// SIMATIC STEP 7 (V5.x) project 0715-19068
// CPU: CPU 315-2 DP
// CPU: CPU 313C
// station: Hardware
// station: Rigid stranding 61/630
// station: P_ADR_BUS
// station: P_ADR_BUS
// station: Hardware
// station: Loader_Cage6_12_18_24
// program: S7 Program
// program: Programma S7
// program: MASTERDRIVES VC(CUVC)
// program: MASTERDRIVES VC(CUVC)
// program: MASTERDRIVES VC(CUVC)
// program: MASTERDRIVES VC(CUVC)
// program: MASTERDRIVES VC(CUVC)
// program: MASTERDRIVES VC(CUVC)
// program: MASTERDRIVES VC(CUVC)
// program: MASTERDRIVES VC(CUVC)
// program: MASTERDRIVES VC(CUVC)
// program: MASTERDRIVES VC(CUVC)

SYMBOL_TABLE
"Drives --> Plc"	DB 1	DB 1	// Drive --> Plc Data Block
"Plc --> Drives"	DB 2	DB 2	// Plc --> Drive Data Block
"Profibus SFC Alarm"	DB 3	DB 3	// Profibus SFC Alarm Data Block
"Take-up traverse"	DB 5	DB 5	// Take-up traverse Data Block
"Take-up"	DB 7	DB 7	// Take-up data block
"Capstan"	DB 9	DB 9	// Capstan data block
"Cage 24"	DB 15	DB 15	// Cage 24 data block
"Cage 24 preforming"	DB 18	DB 18	// Cage 24 preforming data block
"Cage 18"	DB 20	DB 20	// Cage 18 data block
"Cage 18 preforming"	DB 23	DB 23	// Cage 18 preforming data block
"Cage 12"	DB 25	DB 25	// Cage 12 data block
"Cage 12 preforming"	DB 28	DB 28	// Cage 12 preforming data block
"Cage 6"	DB 30	DB 30	// Cage 6 data block
"Pay-off 630"	DB 35	DB 35	// Pay-off 630 data block
"Metercounter"	DB 41	DB 41	// Metercounter data block
"Line"	DB 55	DB 55	// Line data block
"HMI animation"	DB 60	DB 60	// HMI animation data block
"MAP_DI"	DB 91	DB 91	// DIGITAL INPUT MAP
"MAP_DO"	DB 93	DB 93	// DIGITAL OUTPUT MAP
"Db Plc <=> HMI"	DB 100	DB 100	// Db Plc <=> HMI data block
"Count setting"	DB 101	DB 101	// Count setting data block
"FB125"	DB 125	FB 125	// FB125 data block
"DETAIL_DP_DIAG"	FB 125	FB 125
"Alarms Reset"	FC 1	FC 1	// Alarms reset function
"Profibus alarms"	FC 2	FC 2	// Profibus alarms function
"Profibus unit"	FC 3	FC 3	// Profibus unit function
"Take-up traverse alarms"	FC 4	FC 4	// Take-up traverse alarms function
"Take-up traverse unit"	FC 5	FC 5	// Take-up traverse unit function
"Take-up alarms"	FC 6	FC 6	// Take-up alarms function
"Take-up unit"	FC 7	FC 7	// Take-up unit function
"Capstan alarms"	FC 8	FC 8	// Capstan alarms function
"Capstan unit"	FC 9	FC 9	// Capstan unit function
"Door Cage Lock"	FC 10	FC 10	// Door Cage Lock
"Cage common function"	FC 13	FC 13	// Cage common function
"Cage 24 alarms"	FC 14	FC 14	// Cage 24 alarms function
"Cage 24 unit"	FC 15	FC 15	// Cage 24 unit function
"Cage 24 loading fase"	FC 16	FC 16	// Cage 24 loading fase function
"Cage 24 preforming alarm"	FC 17	FC 17	// Cage 24 preforming alarms function
"Cage 24 preforming unit"	FC 18	FC 18	// Cage 24 preforming unit function
"Cage 18 alarms"	FC 19	FC 19	// Cage 18 alarms function
"Cage 18 unit"	FC 20	FC 20	// Cage 18 unit function
"Cage 18 loading fase"	FC 21	FC 21	// Cage 18 loading fase function
"Cage 18 preforming alarm"	FC 22	FC 22	// Cage 18 preforming alarms function
"Cage 18 preforming unit"	FC 23	FC 23	// Cage 18 preforming unit function
"Cage 12 alarms"	FC 24	FC 24	// Cage 12 alarms function
"Cage 12 unit"	FC 25	FC 25	// Cage 12 unit function
"Cage 12 loading fase"	FC 26	FC 26	// Cage 12 loading fase function
"Cage 12 preforming alarm"	FC 27	FC 27	// Cage 12 preforming alarms function
"Cage 12 preforming unit"	FC 28	FC 28	// Cage 12 preforming unit function
"Cage 6 alarms"	FC 29	FC 29	// Cage 6 alarms function
"Cage 6 unit"	FC 30	FC 30	// Cage 6 unit function
"Cage 6 loading fase"	FC 31	FC 31	// Cage 6 loading fase function
"Cage 6 preforming alarms"	FC 32	FC 32	// Cage 6 preforming alarms function
"Cage 6 preforming unit"	FC 33	FC 33	// Cage 6 preforming unit function
"Pay-off 630 alarms"	FC 34	FC 34	// Pay-off 630 alarms function
"Pay-off 630 unit"	FC 35	FC 35	// Pay-off 630 unit function
"Metercounter alarms"	FC 40	FC 40	// Metercounter alarms function
"Metercounter unit"	FC 41	FC 41	// Metercounter unit function
"Common function"	FC 50	FC 50	// Common function
"Hour counter"	FC 51	FC 51	// Hour counter function
"Line alarms"	FC 52	FC 52	// Line alarms function
"Line unit"	FC 53	FC 53	// Line unit function
"Run consent"	FC 54	FC 54	// Run consents function
"Line jog - line run"	FC 55	FC 55	// Line jog - line run function
"Line reference"	FC 56	FC 56	// Line reference function
"Linear speed"	FC 57	FC 57	// Linear speed function
"Missing power supply"	FC 59	FC 59	// Missing power supply function
"HMI animation unit"	FC 60	FC 60	// HMI animation function
"Take-up traverse impulse"	FC 61	FC 61	// Take-up traverse impulses function
"Cage 24 wires insertion"	FC 70	FC 70	// Cage 24 wires insertion function
"Cage 18 wires insertion"	FC 71	FC 71	// Cage 18 wires insertion function
"Cage 12 wires insertion"	FC 72	FC 72	// Cage 12 wires insertion function
"Cage 6 wires insertion"	FC 73	FC 73	// Cage 6 wires insertion function
"Wires break time"	FC 74	FC 74	// Wires break time function
"Bobbins diameter"	FC 79	FC 79	// Bobbins diameter
"Bobbins brake"	FC 80	FC 80	// Bobbins brake
"Rpm increase"	FC 81	FC 81	// Rpm increase
"Map Input Function"	FC 91	FC 91	// Map Input Function
"Map Output Function"	FC 93	FC 93	// Map Output Function
"Increase-decrease"	FC 100	FC 100	// Increase-decrease function
"Flip-Flop"	FC 101	FC 101	// Flip-flop function
"Ramp"	FC 102	FC 102	// Ramp function
"16 Bit Filter"	FC 103	FC 103	// 16 Bit filter function
"Diameter calculation"	FC 105	FC 105	// Diameter calculation function
"Increase-decrease head"	FC 106	FC 106	// Increase-decrease head function
"32 Bit filter"	FC 108	FC 108	// 32 Bit filter function
"Capstan linear speed"	FC 112	FC 112	// Capstan linear speed function
"Bobbins wire management"	FC 113	FC 113	// Bobbins wire management function
"Bobbin diameter calculat"	FC 114	FC 114	// Bobbin diameter calculaton function
"Motor status HMI"	FC 115	FC 115	// Motor status checking for HMI animation function
"Rotation control"	FC 200	FC 200	// Rotation control function
"-126K1:Auxiliary"	I 0.0	BOOL	// Auxiliary on
"-126K4"	I 0.1	BOOL	// Emergency push-buttons
"-175S3"	I 0.2	BOOL	// Cabinet thermo-switch
"-112Q3"	I 0.3	BOOL	// Auxiliary 220v transformer overload
"-108G1:Alarm"	I 0.4	BOOL	// 24DC UPS module battery alarm
"-108G1:Bat ok"	I 0.5	BOOL	// 24DC UPS module battery packs ok
"-116Q1"	I 0.6	BOOL	// Cabinet air fans overload
"E000.7"	I 0.7	BOOL	// Spare
"-119Q1"	I 1.0	BOOL	// Dryer supply overload
"-141R1:T2"	I 1.1	BOOL	// Ac motor drives feeder braking resistor alarm
"-140G1:X104:20"	I 1.2	BOOL	// Ac motor drives feeder dc bus alarm
"-922S3"	I 1.3	BOOL	// Take-up traverse quick left push-buttons main panel
"-922S4"	I 1.4	BOOL	// Take-up traverse quick right push-buttons main panel
"-112Q8"	I 1.5	BOOL	// Take-up 220vac power supply overload
"-109Q7"	I 1.6	BOOL	// Take-up 24vdc power supply overload
"-922S5"	I 1.7	BOOL	// Take-up bobbin increase pull push-button
"-922S6"	I 2.0	BOOL	// Take-up bobbin decrease pull push-button
"-922S7"	I 2.1	BOOL	// Take-up bobbin stop push-buttons
"-922S8"	I 2.2	BOOL	// Take-up bobbin run push-buttons
"-705Q1"	I 2.3	BOOL	// Capstan motor blower overload
"-718S4"	I 2.4	BOOL	// Capstan minimum air pressure pressure-switch
"-718S5"	I 2.5	BOOL	// Capstan motor brake control pressure-switch
"-718B6"	I 2.6	BOOL	// Capstan cable clock open sensor
"-177S6"	I 2.7	BOOL	// Cable block opening selector-switch
"-177S7:Forward"	I 3.0	BOOL	// Capstan forward jog selector-switch
"-177S7:Backward"	I 3.1	BOOL	// Capstan backward jog selector-switch
"-540Q1"	I 3.2	BOOL	// Cage 18 230vac power supply overload
"-109Q11"	I 3.3	BOOL	// Cage 18 24vdc power supply overload
"-505Q2"	I 3.4	BOOL	// Cage 18 loading motor overload
"-505Q1"	I 3.5	BOOL	// Cage 18 motor blower overload
"-507Q2"	I 3.6	BOOL	// Cage 18 preforming motor electric brake overload
"-507Q1"	I 3.7	BOOL	// Cage 18 preforming motor blower overload
"E004.0"	I 4.0	BOOL	// Spare
"-506Q1"	I 4.1	BOOL	// Cage 18 guard blower motor overload
"-440Q1"	I 4.2	BOOL	// Cage 12 230vac power supply overload
"-109Q10"	I 4.3	BOOL	// Cage 12 24vdc power supply overload
"-405Q2"	I 4.4	BOOL	// Cage 12 loading motor overload
"-405Q1"	I 4.5	BOOL	// Cage 12 motor blower overload
"-407Q2"	I 4.6	BOOL	// Cage 12 preforming motor electric brake overload
"-407Q1"	I 4.7	BOOL	// Cage 12 preforming motor blower overload
"E005.0"	I 5.0	BOOL	// Spare
"-406Q1"	I 5.1	BOOL	// Cage 12 guard blower motor overload
"-340Q1"	I 5.2	BOOL	// Cage 6 230vac power supply overload
"-109Q9"	I 5.3	BOOL	// Cage 6 24vdc power supply overload
"-305Q2"	I 5.4	BOOL	// Cage 6 loading motor overload
"-305Q1"	I 5.5	BOOL	// Cage 6 motor blower overload
"E005.6"	I 5.6	BOOL	// Spare
"-306Q1"	I 5.7	BOOL	// Cage 6 guard blower motor overload
"E006.0"	I 6.0	BOOL	// Spare
"E006.1"	I 6.1	BOOL	// Spare
"E006.2"	I 6.2	BOOL	// Spare
"-177S1"	I 6.3	BOOL	// Line stop push-buttons
"-177S2"	I 6.4	BOOL	// Line run push-buttons
"-177S3"	I 6.5	BOOL	// Line jog push-buttons
"-177S4"	I 6.6	BOOL	// Line alarms reset push-buttons
"-177S5"	I 6.7	BOOL	// Hold line speed push-button
"-640Q1"	I 7.0	BOOL	// Cage 24 230VAC supply overload
"-109Q12"	I 7.1	BOOL	// Cage 24 24VDC supply overload
"-605Q2"	I 7.2	BOOL	// Cage 24 loading motor overload
"-605Q1"	I 7.3	BOOL	// Cage 24 motor blower overload
"-607Q2"	I 7.4	BOOL	// Cage 24 preforming motor electric brake overload
"-607Q1"	I 7.5	BOOL	// Cage 24 preforming motor blower overload
"E007.6"	I 7.6	BOOL	// Spare
"-606Q1"	I 7.7	BOOL	// Cage 24 guard  blower motor overload
"-112K1"	I 8.0	BOOL	// Power supply on
"-112K1:66"	I 8.1	BOOL	// Power supply on end of time
"-113G1:4"	I 8.2	BOOL	// 230VAC UPS main failure
"-113G1:3"	I 8.3	BOOL	// 230VAC UPS battery nearly low
"-109Q6"	I 8.4	BOOL	// 24DC aux. feeding overload
"-115Q1"	I 8.5	BOOL	// preforming motor blower and inverter fan supply overload
"-140Q1"	I 8.6	BOOL	// AC motor drive feeder fan overload
"-109Q2"	I 8.7	BOOL	// 24VDC PLC input supply overload
"+MCB06:7"	I 9.0	BOOL	// Cage 6 Loader in stand by zone
"+MCB06:8"	I 9.1	BOOL	// Cage 6 Loader inside cage
"+MCB06:9"	I 9.2	BOOL	// Cage 6 Loader open clamp
"+MCB06:10"	I 9.3	BOOL	// Cage 6 Loader to parcking zone
"+MCB12:7"	I 9.4	BOOL	// Cage 12 Loader in stand by zone
"+MCB12:8"	I 9.5	BOOL	// Cage 12 Loader inside cage
"+MCB12:9"	I 9.6	BOOL	// Cage 12 Loader open clamp
"+MCB12:10"	I 9.7	BOOL	// Cage 12 Loader to parcking zone
"+MCB18:7"	I 10.0	BOOL	// Cage 18 Loader in stand by zone
"+MCB18:8"	I 10.1	BOOL	// Cage 18 Loader inside cage
"+MCB18:9"	I 10.2	BOOL	// Cage 18 Loader open clamp
"+MCB18:10"	I 10.3	BOOL	// Cage 18 Loader to parcking zone
"+MCB24:7"	I 10.4	BOOL	// Cage 24 Loader in stand by zone
"+MCB24:8"	I 10.5	BOOL	// Cage 24 Loader inside cage
"+MCB24:9"	I 10.6	BOOL	// Cage 24 Loader open clamp
"+MCB24:10"	I 10.7	BOOL	// Cage 24 Loader to parcking zone
"E011.0"	I 11.0	BOOL	// Spare
"E011.1"	I 11.1	BOOL	// Spare
"E011.2"	I 11.2	BOOL	// Spare
"E011.3"	I 11.3	BOOL	// Spare
"E011.4"	I 11.4	BOOL	// Spare
"E011.5"	I 11.5	BOOL	// Spare
"E011.6"	I 11.6	BOOL	// Spare
"E011.7"	I 11.7	BOOL	// Spare
"-961S1"	I 32.0	BOOL	// Take-up idle pintle up limit-switch
"-961S2"	I 32.1	BOOL	// Take-up idle pintle down limit-switch
"-961S3"	I 32.2	BOOL	// Take-up driven pintle up limit-switch
"-961S4"	I 32.3	BOOL	// Take-up driven pintle down limit-switch
"-961S5:UP"	I 33.0	BOOL	// Take-up driven pintle up selector-switch
"-961S5:DOWN"	I 33.1	BOOL	// Take-up driven pintle down selector-switch
"-961S7:UP"	I 33.2	BOOL	// Take-up idle pintle up selector-switch
"-961S7:DOWN"	I 33.3	BOOL	// Take-up idle pintle down selector-switch
"-962S1:UP"	I 34.0	BOOL	// Take-up pintles up selector-switches
"-962S1:DOWN"	I 34.1	BOOL	// Take-up pintles down selector-switches
"-962S3:OPEN"	I 34.2	BOOL	// Take-up idle pintle opening selector-switches
"-962S3:CLOSE"	I 34.3	BOOL	// Take-up idle pintle closing selector-switches
"-962S5"	I 35.0	BOOL	// Take-up idle pintle emergency limit-switch
"-962S6"	I 35.1	BOOL	// Take-up driven pintle emergency limit-switch
"-962S7"	I 35.2	BOOL	// Take-up traverse quick left push-buttons local panel
"-962S8"	I 35.3	BOOL	// Take-up traverse quick right push-buttons local panel
"-964S1:Forward"	I 36.0	BOOL	// Take-up bobbin forward jog selector-switch
"-964S1:Backward"	I 36.1	BOOL	// Take-up bobbin backward jog selector-switch
"-964B3"	I 36.2	BOOL	// Take-up traverse translation zero point sensor
"-964B4"	I 36.3	BOOL	// Take-up traverse inversion delay sensor
"-941Q2"	I 37.0	BOOL	// Take-up bobbin motor electric brake overload
"-945Q2"	I 37.1	BOOL	// Take-up traverse motor blower overload
"-944Q1"	I 37.2	BOOL	// Take-up ac motors overload
"-945Q1"	I 37.3	BOOL	// Take-up bobbin motor blower overload
"-661S1"	I 42.0	BOOL	// Cage 24 loading line presence of air pressure-switch
"-661S2"	I 42.1	BOOL	// Cage 24 brake control pressure-switch
"-661S3"	I 42.2	BOOL	// Cage 24 minimum air pressure pressure-switch
"-661S4"	I 42.3	BOOL	// Cage 24 piston engaged into cage limit-switch
"-661S5"	I 42.4	BOOL	// Cage 24 piston disingaged out of cage limit-switch
"-661S6"	I 42.5	BOOL	// Cage 24 loading motor engaged sensor
"-661S7"	I 42.6	BOOL	// Cage 24 loading motor disengaged sensor
"-661S8"	I 42.7	BOOL	// Cage 24 air pipe  limit-switch
"-662B1"	I 43.0	BOOL	// Cage 24 presence of bobbin photocell -loading-
"-662B2"	I 43.1	BOOL	// Cage 24 loading stop photocell
"-662S3"	I 43.2	BOOL	// Cage 24 break of wire from ring
"-686Y1"	I 43.3	BOOL	// Cage 24 front door limit-switch
"-662S5"	I 43.4	BOOL	// Cage 24 rear door limit-switches
"-662S6"	I 43.5	BOOL	// Cage 24 front guard open limit-switch
"-662B7"	I 43.6	BOOL	// Cage 24 front guard closed sensor
"-662B8"	I 43.7	BOOL	// Cage 24 guard presence of man photocell
"-663S1"	I 44.0	BOOL	// Cage 24 line stop push-button
"-663S2"	I 44.1	BOOL	// Cage 24 line jog push-button
"-663S3"	I 44.2	BOOL	// Cage 24 loading run push-button
"-663S4"	I 44.3	BOOL	// Cage 24 alarms reset push-button
"-663S5:CLOSING"	I 44.4	BOOL	// Cage 24 guard closing selector-switch
"-663S5:OPENING"	I 44.5	BOOL	// Cage 24 guard opening selector-switch
"-663S7:CLOSING"	I 44.6	BOOL	// Cage 24 pintles closing selector-switch
"-663S7:OPENING"	I 44.7	BOOL	// Cage 24 pintles opening selector-switch
"-664S1:CLOSING"	I 45.0	BOOL	// Cage 24 pintles locking system closing selector-switch
"-664S1:OPENING"	I 45.1	BOOL	// Cage 24 pintles locking system opening selector-switch
"E045.2"	I 45.2	BOOL	// Spare
"E045.3"	I 45.3	BOOL	// Spare
"E045.4"	I 45.4	BOOL	// Spare
"E045.5"	I 45.5	BOOL	// Spare
"-664S7"	I 45.6	BOOL	// Cage 24 loading insertion push-button
"E045.7"	I 45.7	BOOL	// Spare
"E046.0"	I 46.0	BOOL	// Spare
"E046.1"	I 46.1	BOOL	// Spare
"E046.2"	I 46.2	BOOL	// Spare
"E046.3"	I 46.3	BOOL	// Spare
"E046.4"	I 46.4	BOOL	// Spare
"E046.5"	I 46.5	BOOL	// Spare
"-688Y8"	I 46.6	BOOL	// Cage 24 preforming guard limit-switch
"-665S8"	I 46.7	BOOL	// Cage 24 preforming brake release push-button
"-666S1"	I 47.0	BOOL	// Cage 24 preforming line stop push-button
"-666S2"	I 47.1	BOOL	// Cage 24 preforming line jog push-button
"-667B1"	I 47.2	BOOL	// Cage 24 bobbin 1 break of wire and diameter calculation
"-667B2"	I 47.3	BOOL	// Cage 24 bobbin 2 break of wire
"-667B3"	I 47.4	BOOL	// Cage 24 bobbin 3 break of wire
"-667B4"	I 47.5	BOOL	// Cage 24 bobbin 4 break of wire
"-667B5"	I 47.6	BOOL	// Cage 24 bobbin 5 break of wire
"-667B6"	I 47.7	BOOL	// Cage 24 bobbin 6 break of wire
"-667B7"	I 48.0	BOOL	// Cage 24 bobbin 7 break of wire
"-667B8"	I 48.1	BOOL	// Cage 24 bobbin 8 break of wire
"-668B1"	I 48.2	BOOL	// Cage 24 bobbin 9 break of wire
"-668B2"	I 48.3	BOOL	// Cage 24 bobbin 10 break of wire
"-668B3"	I 48.4	BOOL	// Cage 24 bobbin 11 break of wire
"-668B4"	I 48.5	BOOL	// Cage 24 bobbin 12 break of wire
"-668B5"	I 48.6	BOOL	// Cage 24 bobbin 13 break of wire
"-668B6"	I 48.7	BOOL	// Cage 24 bobbin 14 break of wire
"-668B7"	I 49.0	BOOL	// Cage 24 bobbin 15 break of wire
"-668B8"	I 49.1	BOOL	// Cage 24 bobbin 16 break of wire
"-669B1"	I 49.2	BOOL	// Cage 24 bobbin 17 break of wire
"-669B2"	I 49.3	BOOL	// Cage 24 bobbin 18 break of wire
"-669B3"	I 49.4	BOOL	// Cage 24 bobbin 19 break of wire
"-669B4"	I 49.5	BOOL	// Cage 24 bobbin 20 break of wire
"-669B5"	I 49.6	BOOL	// Cage 24 bobbin 21 break of wire
"-669B6"	I 49.7	BOOL	// Cage 24 bobbin 22 break of wire
"-669B7"	I 50.0	BOOL	// Cage 24 bobbin 23 break of wire
"-669B8"	I 50.1	BOOL	// Cage 24 bobbin 24 break of wire
"-670S1"	I 50.2	BOOL	// Cage 24 bobbin brakes air tank pressure switch
"-670S2"	I 50.3	BOOL	// Cage 24 line 1 pintles open
"-670S3"	I 50.4	BOOL	// Cage 24 line 2 pintles open
"-670S4"	I 50.5	BOOL	// Cage 24 line 3 pintles open
"E050.6"	I 50.6	BOOL	// Spare
"E050.7"	I 50.7	BOOL	// Spare
"E051.0"	I 51.0	BOOL	// Spare
"E051.1"	I 51.1	BOOL	// Spare
"E051.2"	I 51.2	BOOL	// Spare
"E051.3"	I 51.3	BOOL	// Spare
"E051.4"	I 51.4	BOOL	// Spare
"E051.5"	I 51.5	BOOL	// Spare
"E051.6"	I 51.6	BOOL	// Spare
"E051.7"	I 51.7	BOOL	// Spare
"-561S1"	I 52.0	BOOL	// Cage 18 loading line presence of air pressure-switch
"-561S2"	I 52.1	BOOL	// Cage 18 brake control pressure-switch
"-561S3"	I 52.2	BOOL	// Cage 18 minimum air pressure pressure-switch
"-561S4"	I 52.3	BOOL	// Cage 18 piston engaged in cage limit-switch
"-561S5"	I 52.4	BOOL	// Cage 18 piston disengaged from cage limit-switch
"-561B6"	I 52.5	BOOL	// Cage 18 loading motor engaged sensor
"-561B7"	I 52.6	BOOL	// Cage 18 loading motor disengaged sensor
"-561S8"	I 52.7	BOOL	// Cage 18 air pipe limit-switch
"-562B1"	I 53.0	BOOL	// Cage 18 presence of bobbin photocell -loading-
"-562B2"	I 53.1	BOOL	// Cage 18 loading stop photocell
"-562S3"	I 53.2	BOOL	// Cage 18 break of wire from ring
"-586Y1"	I 53.3	BOOL	// Cage 18 front door limit-switch
"-562S5"	I 53.4	BOOL	// Cage 18 rear doors limit-switches
"-562S6"	I 53.5	BOOL	// Cage 18 front guard open limit-switch
"-562B7"	I 53.6	BOOL	// Cage 18 front guard closed sensor
"-562B8"	I 53.7	BOOL	// Cage 18 guard presence of man photocell
"-563S1"	I 54.0	BOOL	// Cage 18 line stop push-button
"-563S2"	I 54.1	BOOL	// Cage 18 line jog push-button
"-563S3"	I 54.2	BOOL	// Cage 18 loading run push-button
"-563S4"	I 54.3	BOOL	// Cage 18 alarms reset push-button
"-563S5:CLOSING"	I 54.4	BOOL	// Cage 18 guard closing selector-switch
"-563S5:OPENING"	I 54.5	BOOL	// Cage 18 guard opening selector-switch
"-563S7:CLOSING"	I 54.6	BOOL	// Cage 18 pintles closing selector-switch
"-563S7:OPENING"	I 54.7	BOOL	// Cage 18 pintles opening selector-switch
"-564S1:CLOSING"	I 55.0	BOOL	// Cage 18 pintles locking system closing selector-switch
"-563S1:OPENING"	I 55.1	BOOL	// Cage 18 pintles locking system opening selector-switch
"E055.2"	I 55.2	BOOL	// Spare
"E055.3"	I 55.3	BOOL	// Spare
"E055.4"	I 55.4	BOOL	// Spare
"E055.5"	I 55.5	BOOL	// Spare
"-564S7"	I 55.6	BOOL	// Cage 18 loading insertion push-button
"E055.7"	I 55.7	BOOL	// Spare
"E056.0"	I 56.0	BOOL	// Spare
"E056.1"	I 56.1	BOOL	// Spare
"E056.2"	I 56.2	BOOL	// Spare
"E056.3"	I 56.3	BOOL	// Spare
"-565B5"	I 56.4	BOOL	// Cage 18 Loader Locked
"-565B6"	I 56.5	BOOL	// Cage 18 Loader UnLocked
"-588Y8"	I 56.6	BOOL	// Cage 18 preforming guard limit-switch
"-565S8"	I 56.7	BOOL	// Cage 18 preforming brake release push-button
"-566S1"	I 57.0	BOOL	// Cage 18 preforming line stop push-button
"-566S2"	I 57.1	BOOL	// Cage 18 preforming line jog push-button
"-567B1"	I 57.2	BOOL	// Cage 18 bobbin 1 break of wire and diameter calculation
"-567B2"	I 57.3	BOOL	// Cage 18 bobbin 2 break of wire
"-567B3"	I 57.4	BOOL	// Cage 18 bobbin 3 break of wire
"-567B4"	I 57.5	BOOL	// Cage 18 bobbin 4 break of wire
"-567B5"	I 57.6	BOOL	// Cage 18 bobbin 5 break of wire
"-567B6"	I 57.7	BOOL	// Cage 18 bobbin 6 break of wire
"-567B7"	I 58.0	BOOL	// Cage 18 bobbin 7 break of wire
"-567B8"	I 58.1	BOOL	// Cage 18 bobbin 8 break of wire
"-568B1"	I 58.2	BOOL	// Cage 18 bobbin 9 break of wire
"-568B2"	I 58.3	BOOL	// Cage 18 bobbin 10 break of wire
"-568B3"	I 58.4	BOOL	// Cage 18 bobbin 11 break of wire
"-568B4"	I 58.5	BOOL	// Cage 18 bobbin 12 break of wire
"-568B5"	I 58.6	BOOL	// Cage 18 bobbin 13 break of wire
"-568B6"	I 58.7	BOOL	// Cage 18 bobbin 14 break of wire
"-568B7"	I 59.0	BOOL	// Cage 18 bobbin 15 break of wire
"-568B8"	I 59.1	BOOL	// Cage 18 bobbin 16 break of wire
"-569B1"	I 59.2	BOOL	// Cage 18 bobbin 17 break of wire
"-569B2"	I 59.3	BOOL	// Cage 18 bobbin 18 break of wire
"-569S3"	I 59.4	BOOL	// Cage 18 bobbin brakes air tank minimum pressure pressure-switch
"-569S4"	I 59.5	BOOL	// Cage 18 line 1 pintles open
"-569S5"	I 59.6	BOOL	// Cage 18 line 2 pintles open
"-569S6"	I 59.7	BOOL	// Cage 18 line 3 pintles open
"-461S1"	I 62.0	BOOL	// Cage 12 loading line presence of air pressure-switch
"-461S2"	I 62.1	BOOL	// Cage 12 brake control pressure-switch
"-461S3"	I 62.2	BOOL	// Cage 12 minimum air pressure pressure-switch
"-461S4"	I 62.3	BOOL	// Cage 12 piston engaged in cage limit-switch
"-461S5"	I 62.4	BOOL	// Cage 12 piston disengaged from cage limit-switch
"-461B6"	I 62.5	BOOL	// Cage 12 loading motor engaged sensor
"-461B7"	I 62.6	BOOL	// Cage 12 loading motor disengaged sensor
"-461S8"	I 62.7	BOOL	// Cage 12 air pipe limit-switch
"-462B1"	I 63.0	BOOL	// Cage 12 presence of bobbin photocell -loading-
"-462B2"	I 63.1	BOOL	// Cage 12 loading stop photocell
"-462S3"	I 63.2	BOOL	// Cage 12 break of wire from ring
"-486Y1"	I 63.3	BOOL	// Cage 12 front door limit-switch
"-462S5"	I 63.4	BOOL	// Cage 12 rear doors limit-switches
"-462S6"	I 63.5	BOOL	// Cage 12 front guard open limit-switch
"-462B7"	I 63.6	BOOL	// Cage 12 front guard closed sensor
"-462B8"	I 63.7	BOOL	// Cage 12 guard presence of man photocell
"-463S1"	I 64.0	BOOL	// Cage 12 line stop push-button
"-463S2"	I 64.1	BOOL	// Cage 12 line jog push-button
"-463S3"	I 64.2	BOOL	// Cage 12 loading run push-button
"-463S4"	I 64.3	BOOL	// Cage 12 alarms reset push-button
"-463S5:CLOSING"	I 64.4	BOOL	// Cage 12 guard closing selector-switch
"-463S5:OPENING"	I 64.5	BOOL	// Cage 12 guard opening selector-switch
"-463S7:CLOSING"	I 64.6	BOOL	// Cage 12 pintles closing selector-switch
"-463S7:OPENING"	I 64.7	BOOL	// Cage 12 pintles opening selector-switch
"-464S1:CLOSING"	I 65.0	BOOL	// Cage 12 pintles locking system closing selector-switch
"-464S1:OPENING"	I 65.1	BOOL	// Cage 12 pintles locking system opening selector-switch
"E065.2"	I 65.2	BOOL	// Spare
"E065.3"	I 65.3	BOOL	// Spare
"E065.4"	I 65.4	BOOL	// Spare
"E065.5"	I 65.5	BOOL	// Spare
"-464S7"	I 65.6	BOOL	// Cage 12 loading insertion push-button
"E065.7"	I 65.7	BOOL	// Spare
"E066.0"	I 66.0	BOOL	// Spare
"E066.1"	I 66.1	BOOL	// Spare
"E066.2"	I 66.2	BOOL	// Spare
"E066.3"	I 66.3	BOOL	// Spare
"E066.4"	I 66.4	BOOL	// Spare
"E066.5"	I 66.5	BOOL	// Spare
"-488Y8"	I 66.6	BOOL	// Cage 12 preforming guard limit-switch
"-465S8"	I 66.7	BOOL	// Cage 12 preforming brake release push-button
"-466S1"	I 67.0	BOOL	// Cage 12 preforming line stop push-button
"-466S2"	I 67.1	BOOL	// Cage 12 preforming line jog push-button
"-467B1"	I 67.2	BOOL	// Cage 12 bobbin 1 break of wire and diameter calculation
"-467B2"	I 67.3	BOOL	// Cage 12 bobbin 2 break of wire
"-467B3"	I 67.4	BOOL	// Cage 12 bobbin 3 break of wire
"-467B4"	I 67.5	BOOL	// Cage 12 bobbin 4 break of wire
"-467B5"	I 67.6	BOOL	// Cage 12 bobbin 5 break of wire
"-467B6"	I 67.7	BOOL	// Cage 12 bobbin 6 break of wire
"-467B7"	I 68.0	BOOL	// Cage 12 bobbin 7 break of wire
"-467B8"	I 68.1	BOOL	// Cage 12 bobbin 8 break of wire
"-468B1"	I 68.2	BOOL	// Cage 12 bobbin 9 break of wire
"-468B2"	I 68.3	BOOL	// Cage 12 bobbin 10 break of wire
"-468B3"	I 68.4	BOOL	// Cage 12 bobbin 11 break of wire
"-468B4"	I 68.5	BOOL	// Cage 12 bobbin 12 break of wire
"-468S5"	I 68.6	BOOL	// Cage 12 bobbin brakes air tank minimum pressure pressure-switch
"-468S6"	I 68.7	BOOL	// Cage 12 line 1 pintles open
"-468S7"	I 69.0	BOOL	// Cage 12 line 2 pintles open
"-468S8"	I 69.1	BOOL	// Cage 12 line 3 pintles open
"-475S1/S1A"	I 69.2	BOOL	// Cage 12 loader unlocked
"-475S2/S2A"	I 69.3	BOOL	// Cage 12 loader locked
"E069.4"	I 69.4	BOOL	// Spare
"E069.5"	I 69.5	BOOL	// Spare
"E069.6"	I 69.6	BOOL	// Spare
"E069.7"	I 69.7	BOOL	// Spare
"-361S1"	I 72.0	BOOL	// Cage 6 loading line presence of air pressure-switch
"-361S2"	I 72.1	BOOL	// Cage 6 brake control pressure-switch
"-361S3"	I 72.2	BOOL	// Cage 6 minimum air pressure pressure-switch
"-361S4"	I 72.3	BOOL	// Cage 6 piston engaged in cage limit-switch
"-361S5"	I 72.4	BOOL	// Cage 6 piston disengaged from cage limit-switch
"-361B6"	I 72.5	BOOL	// Cage 6 loading motor engaged sensor
"-361B7"	I 72.6	BOOL	// Cage 6 loading motor disengaged sensor
"-361S8"	I 72.7	BOOL	// Cage 6 air pipe limit-switch
"-361B1"	I 73.0	BOOL	// Cage 6 presence of bobbin photocell -loading-
"-362B2"	I 73.1	BOOL	// Cage 6 loading stop photocell
"-362S3"	I 73.2	BOOL	// Cage 6 break of wire from ring
"-386Y1"	I 73.3	BOOL	// Cage 6 front door limit-switch
"-362S5"	I 73.4	BOOL	// Cage 6 rear doors limit-switches
"-362S6"	I 73.5	BOOL	// Cage 6 front guard open limit-switch
"-362B7"	I 73.6	BOOL	// Cage 6 front guard closed sensor
"-362B8"	I 73.7	BOOL	// Cage 6 guard presence of man photocell
"-363S1"	I 74.0	BOOL	// Cage 6 line stop push-button
"-363S2"	I 74.1	BOOL	// Cage 6 line jog push-button
"-363S3"	I 74.2	BOOL	// Cage 6 loading run push-button
"-363S4"	I 74.3	BOOL	// Cage 6 alarms reset push-button
"-363S5:CLOSING"	I 74.4	BOOL	// Cage 6 guard closing selector-switch
"-363S5:OPENING"	I 74.5	BOOL	// Cage 6 guard opening selector-switch
"-363S7:CLOSING"	I 74.6	BOOL	// Cage 6 pintles closing selector-switch
"-363S7:OPENING"	I 74.7	BOOL	// Cage 6 pintles opening selector-switch
"-364S1:Closing"	I 75.0	BOOL	// Cage 6 pintles locking system closing selector-switch
"-364S1:Opening"	I 75.1	BOOL	// Cage 6 pintles locking system opening selector-switch
"E075.2"	I 75.2	BOOL	// Spare
"E075.3"	I 75.3	BOOL	// Spare
"E075.4"	I 75.4	BOOL	// Spare
"E075.5"	I 75.5	BOOL	// Spare
"-364S7"	I 75.6	BOOL	// Cage 6 loading insertion push-button
"E075.7"	I 75.7	BOOL	// Spare
"E076.0"	I 76.0	BOOL	// Spare
"E076.1"	I 76.1	BOOL	// Spare
"E076.2"	I 76.2	BOOL	// Spare
"E076.3"	I 76.3	BOOL	// Spare
"E076.4"	I 76.4	BOOL	// Spare
"E076.5"	I 76.5	BOOL	// Spare
"-388Y8"	I 76.6	BOOL	// Cage 6 preforming guard limit-switch
"-365S"	I 76.7	BOOL	// Cage 6 preforming line stop push-button
"-366S1"	I 77.0	BOOL	// Cage 6 preforming line jog push-button
"-367B1"	I 77.1	BOOL	// Cage 6 bobbin 1 break of wire and diameter calculation
"-367B2"	I 77.2	BOOL	// Cage 6 bobbin 2 break of wire
"-367B3"	I 77.3	BOOL	// Cage 6 bobbin 3 break of wire
"-367B4"	I 77.4	BOOL	// Cage 6 bobbin 4 break of wire
"-367B5"	I 77.5	BOOL	// Cage 6 bobbin 5 break of wire
"-367B6"	I 77.6	BOOL	// Cage 6 bobbin 6 break of wire
"-367S7"	I 77.7	BOOL	// Cage 6 bobbin brakes air tank minimum pressure pressure-switch
"-367S8"	I 78.0	BOOL	// Cage 6 line 1 pintles open
"-368S1"	I 78.1	BOOL	// Cage 6 line 2 pintles open
"-368S2"	I 78.2	BOOL	// Cage 6 line 3 pintles open
"E078.3"	I 78.3	BOOL	// Spare
"E078.4"	I 78.4	BOOL	// Spare
"E078.5"	I 78.5	BOOL	// Spare
"E078.6"	I 78.6	BOOL	// Spare
"-375S1"	I 78.7	BOOL	// Central Pay-off 630 pintle close selector-switch
"-375B1"	I 79.0	BOOL	// Central Pay-off 630 break of wire sensor
"-375S3"	I 79.1	BOOL	// Central Pay-off 630 main air minimum pressure-switch
"-375S4"	I 79.2	BOOL	// Central Pay-off 630 line stop push-button
"-375S5"	I 79.3	BOOL	// Central Pay-off 630 break release push-button
"-374S7/S7A"	I 79.4	BOOL	// Cage 6 loader unlocked
"-375S7/S7A"	I 79.5	BOOL	// Cage 6 loader locked
"E079.6"	I 79.6	BOOL	// Spare
"E079.7"	I 79.7	BOOL	// Spare
"EB43"	IB 43	BYTE	// Cage 24 digital input
"EB53"	IB 53	BYTE	// Cage 18 digital input
"EB63"	IB 63	BYTE	// Cage 12 digital input
"EB73"	IB 73	BYTE	// Cage 6 digital input
"M1.0"	M 1.0	BOOL	// Clock 0,1 Sec
"M1.1"	M 1.1	BOOL	// Clock 0,2 Sec
"M1.2"	M 1.2	BOOL	// Clock 0,4 Sec
"M1.3"	M 1.3	BOOL	// Clock 0,5 Sec
"M1.4"	M 1.4	BOOL	// Clock 0,8 Sec
"M1.5"	M 1.5	BOOL	// Clock 1,0 Sec
"M1.6"	M 1.6	BOOL	// Clock 1,6 Sec
"M1.7"	M 1.7	BOOL	// Clock 2,0 Sec
"M2.0"	M 2.0	BOOL	// 100 ms impulse
"M2.1"	M 2.1	BOOL	// 200 ms impulse
"M2.2"	M 2.2	BOOL	// 400 ms impulse
"M2.3"	M 2.3	BOOL	// 500 ms impulse
"M2.4"	M 2.4	BOOL	// 800 ms impulse
"M2.5"	M 2.5	BOOL	// 1 s impulse
"M2.6"	M 2.6	BOOL	// 1,6 s impulse
"M2.7"	M 2.7	BOOL	// 2 s impulse
"M3.0"	M 3.0	BOOL	// 100 ms positive edge
"M3.1"	M 3.1	BOOL	// 200 ms positive edge
"M3.2"	M 3.2	BOOL	// 400 ms positive edge
"M3.3"	M 3.3	BOOL	// 500 ms positive edge
"M3.4"	M 3.4	BOOL	// 800 ms positive edge
"M3.5"	M 3.5	BOOL	// 1 s positive edge
"M3.6"	M 3.6	BOOL	// 1,6 s positive edge
"M3.7"	M 3.7	BOOL	// 2 s positive edge
"block"	M 7.0	BOOL	// Маркер блокировки аварий
"M10.1"	M 10.1	BOOL	// Take-up traverse direction
"M10.2"	M 10.2	BOOL	// Take-up traverse inversion delay
"M10.3"	M 10.3	BOOL	// Take-up traverse inversion delay sensor edge positive
"M10.4"	M 10.4	BOOL	// Take-up traverse inversion edge positive
"M11.0"	M 11.1	BOOL	// 1=Door_Lock, 0=Door_UnLock
"M12.0"	M 12.0	BOOL	// Auxiliary ramp
"M12.1"	M 12.1	BOOL	// Auxiliary ramp
"M12.2"	M 12.2	BOOL	// Auxiliary ramp
"M12.3"	M 12.3	BOOL	// Auxiliary ramp
"M12.4"	M 12.4	BOOL	// Auxiliary ramp
"M12.5"	M 12.5	BOOL	// Auxiliary ramp
"M12.6"	M 12.6	BOOL	// Auxiliary ramp
"M12.7"	M 12.7	BOOL	// Auxiliary ramp
"M13.1"	M 13.1	BOOL	// Take-up increase-decrease auxiliary
"M14.0"	M 14.0	BOOL	// Cage 6 Flip-flop auxiliary flag 1
"M14.1"	M 14.1	BOOL	// Cage 6 Flip-flop auxiliary flag 2
"M14.2"	M 14.2	BOOL	// Cage 6 flip-flop output for loading on-off
"M14.3"	M 14.3	BOOL	// Cage 6 call for loading on
"M14.4"	M 14.4	BOOL	// Cage 6 call for loading off
"M15.0"	M 15.0	BOOL	// Cage 12 Flip-flop auxiliary flag 1
"M15.1"	M 15.1	BOOL	// Cage 12 Flip-flop auxiliary flag 2
"M15.2"	M 15.2	BOOL	// Cage 12 flip-flop output for loading on-off
"M15.3"	M 15.3	BOOL	// Cage 12 call for loading on
"M15.4"	M 15.4	BOOL	// Cage 12 call for loading off
"M16.0"	M 16.0	BOOL	// Cage 18 Flip-flop auxiliary flag 1
"M16.1"	M 16.1	BOOL	// Cage 18 Flip-flop auxiliary flag 2
"M16.2"	M 16.2	BOOL	// Cage 18 flip-flop output for loading on-off
"M16.3"	M 16.3	BOOL	// Cage 18 call for loading on
"M16.4"	M 16.4	BOOL	// Cage 18 call for loading off
"M017.0"	M 17.0	BOOL	// Cage 24 Flip-flop auxiliary flag 1
"M017.1"	M 17.1	BOOL	// Cage 24 Flip-flop auxiliary flag 2
"M017.2"	M 17.2	BOOL	// Cage 24 flip-flop output for loading on-off
"M017.3"	M 17.3	BOOL	// Cage 24 call for loading on
"M017.4"	M 17.4	BOOL	// Cage 24 call for loading off
"M18.1"	M 18.1	BOOL	// Cage 6 bobbin 1 impulse rlc edge
"M18.2"	M 18.2	BOOL	// Cage 12 bobbin 1 impulse rlc edge
"M18.3"	M 18.3	BOOL	// Cage 18 bobbin 1 impulse rlc edge
"M18.4"	M 18.4	BOOL	// Cage 24 bobbin 1 impulse rlc edge
"M19.0"	M 19.0	BOOL	// Pay-off 630 bobbin impulse rlc edge
"M20.0"	M 20.0	BOOL	// Loading run from One o more cages
"M20.2"	M 20.2	BOOL	// Line jog push-buttons of one o more cage
"M20.3"	M 20.3	BOOL	// Loading run push-button of one o more cage
"M20.4"	M 20.4	BOOL	// Preforming line jog push-button of one o more cage
"M20.6"	M 20.6	BOOL	// Loading run from one of cage with piston disengaged
"M20.7"	M 20.7	BOOL	// Preforming line stop global push-buttons
"M21.0"	M 21.0	BOOL	// Line stop global push-buttons
"M21.1"	M 21.1	BOOL	// Not loading run from all cage
"M21.3"	M 21.3	BOOL	// Loading run from one of cage on with piston disengaged
"M30.0"	M 30.0	BOOL	// PLC<-->OP Comunication control
"M30.1"	M 30.1	BOOL	// Alarms Reset
"M50.0"	M 50.0	BOOL	// Cage 6 bobbins wire break control insertion
"M50.1"	M 50.1	BOOL	// Aux. M50.2
"M50.2"	M 50.2	BOOL	// Cage 6 bobbin 1 wire break on
"M50.3"	M 50.3	BOOL	// Cage 6 bobbin 1 counter increase auxiliary
"M50.4"	M 50.4	BOOL	// Aux. M50.5
"M50.5"	M 50.5	BOOL	// Cage 6 bobbin 2 wire break on
"M50.6"	M 50.6	BOOL	// Cage 6 bobbin 2 counter increase auxiliary
"M50.7"	M 50.7	BOOL	// Aux. M51.0
"M51.0"	M 51.0	BOOL	// Cage 6 bobbin 3 wire break on
"M51.1"	M 51.1	BOOL	// Cage 6 bobbin 3 counter increase auxiliary
"M51.2"	M 51.2	BOOL	// Aux. M51.3
"M51.3"	M 51.3	BOOL	// Cage 6 bobbin 4 wire break on
"M51.4"	M 51.4	BOOL	// Cage 6 bobbin 4 counter increase auxiliary
"M51.5"	M 51.5	BOOL	// Aux. M51.6
"M51.6"	M 51.6	BOOL	// Cage 6 bobbin 5 wire break on
"M51.7"	M 51.7	BOOL	// Cage 6 bobbin 5 counter increase auxiliary
"M52.0"	M 52.0	BOOL	// Aux. M52.1
"M52.1"	M 52.1	BOOL	// Cage 6 bobbin 6 wire break on
"M52.2"	M 52.2	BOOL	// Cage 6 bobbin 6 counter increase auxiliary
"M60.0"	M 60.0	BOOL	// Cage 12 bobbins wire break control insertion
"M60.1"	M 60.1	BOOL	// Aux. M60.2
"M60.2"	M 60.2	BOOL	// Cage 12 bobbin 1 wire break on
"M60.3"	M 60.3	BOOL	// Cage 12 bobbin 1 counter increase auxiliary
"M60.4"	M 60.4	BOOL	// Aux. M60.5
"M60.5"	M 60.5	BOOL	// Cage 12 bobbin 2 wire break on
"M60.6"	M 60.6	BOOL	// Cage 12 bobbin 2 counter increase auxiliary
"M60.7"	M 60.7	BOOL	// Aux. M61.0
"M61.0"	M 61.0	BOOL	// Cage 12 bobbin 3 wire break on
"M61.1"	M 61.1	BOOL	// Cage 12 bobbin 3 counter increase auxiliary
"M61.2"	M 61.2	BOOL	// Aux. M61.3
"M61.3"	M 61.3	BOOL	// Cage 12 bobbin 4 wire break on
"M61.4"	M 61.4	BOOL	// Cage 12 bobbin 4 counter increase auxiliary
"M61.5"	M 61.5	BOOL	// Aux. M61.6
"M61.6"	M 61.6	BOOL	// Cage 12 bobbin 5 wire break on
"M61.7"	M 61.7	BOOL	// Cage 12 bobbin 5 counter increase auxiliary
"M62.0"	M 62.0	BOOL	// Aux. M62.1
"M62.1"	M 62.1	BOOL	// Cage 12 bobbin 6 wire break on
"M62.2"	M 62.2	BOOL	// Cage 12 bobbin 6 counter increase auxiliary
"M62.3"	M 62.3	BOOL	// Aux. M62.4
"M62.4"	M 62.4	BOOL	// Cage 12 bobbin 7 wire break on
"M62.5"	M 62.5	BOOL	// Cage 12 bobbin 7 counter increase auxiliary
"M62.6"	M 62.6	BOOL	// Aux. M62.7
"M62.7"	M 62.7	BOOL	// Cage 12 bobbin 8 wire break on
"M63.0"	M 63.0	BOOL	// Cage 12 bobbin 8 counter increase auxiliary
"M63.1"	M 63.1	BOOL	// Aux. M63.2
"M63.2"	M 63.2	BOOL	// Cage 12 bobbin 9 wire break on
"M63.3"	M 63.3	BOOL	// Cage 12 bobbin 9 counter increase auxiliary
"M63.4"	M 63.4	BOOL	// Aux. M63.5
"M63.5"	M 63.5	BOOL	// Cage 12 bobbin 10 wire break on
"M63.6"	M 63.6	BOOL	// Cage 12 bobbin 10 counter increase auxiliary
"M63.7"	M 63.7	BOOL	// Aux. M64.0
"M64.0"	M 64.0	BOOL	// Cage 12 bobbin 11 wire break on
"M64.1"	M 64.1	BOOL	// Cage 12 bobbin 11 counter increase auxiliary
"M64.2"	M 64.2	BOOL	// Aux. M64.3
"M64.3"	M 64.3	BOOL	// Cage 12 bobbin 12 wire break on
"M64.4"	M 64.4	BOOL	// Cage 12 bobbin 12 counter increase auxiliary
"M70.0"	M 70.0	BOOL	// Cage 18 bobbins wire break control insertion
"M70.1"	M 70.1	BOOL	// Aux. M70.2
"M70.2"	M 70.2	BOOL	// Cage 18 bobbin 1 wire break on
"M70.3"	M 70.3	BOOL	// Cage 18 bobbin 1 counter increase auxiliary
"M70.4"	M 70.4	BOOL	// Aux. M70.5
"M70.5"	M 70.5	BOOL	// Cage 18 bobbin 2 wire break on
"M70.6"	M 70.6	BOOL	// Cage 18 bobbin 2 counter increase auxiliary
"M70.7"	M 70.7	BOOL	// Aux. M71.7
"M71.0"	M 71.0	BOOL	// Cage 18 bobbin 3 wire break on
"M71.1"	M 71.1	BOOL	// Cage 18 bobbin 3 counter increase auxiliary
"M71.2"	M 71.2	BOOL	// Aux. M71.3
"M71.3"	M 71.3	BOOL	// Cage 18 bobbin 4 wire break on
"M71.4"	M 71.4	BOOL	// Cage 18 bobbin 4 counter increase auxiliary
"M71.5"	M 71.5	BOOL	// Aux. M71.6
"M71.6"	M 71.6	BOOL	// Cage 18 bobbin 5 wire break on
"M71.7"	M 71.7	BOOL	// Cage 18 bobbin 5 counter increase auxiliary
"M72.0"	M 72.0	BOOL	// Aux. M72.1
"M72.1"	M 72.1	BOOL	// Cage 18 bobbin 6 wire break on
"M72.2"	M 72.2	BOOL	// Cage 18 bobbin 6 counter increase auxiliary
"M72.3"	M 72.3	BOOL	// Aux. M72.4
"M72.4"	M 72.4	BOOL	// Cage 18 bobbin 7 wire break on
"M72.5"	M 72.5	BOOL	// Cage 18 bobbin 7 counter increase auxiliary
"M72.6"	M 72.6	BOOL	// Aux. M72.7
"M72.7"	M 72.7	BOOL	// Cage 18 bobbin 8 wire break on
"M73.1"	M 73.1	BOOL	// Aux. M73.2
"M73.2"	M 73.2	BOOL	// Cage 18 bobbin 9 wire break on
"M73.3"	M 73.3	BOOL	// Cage 18 bobbin 9 counter increase auxiliary
"M73.4"	M 73.4	BOOL	// Aux. M73.5
"M73.5"	M 73.5	BOOL	// Cage 18 bobbin 10 wire break on
"M73.6"	M 73.6	BOOL	// Cage 18 bobbin 10 counter increase auxiliary
"M73.7"	M 73.7	BOOL	// Aux. M74.0
"M74.0"	M 74.0	BOOL	// Cage 18 bobbin 11 wire break on
"M74.2"	M 74.2	BOOL	// Aux. M74.3
"M74.3"	M 74.3	BOOL	// Cage 18 bobbin 12 wire break on
"M74.4"	M 74.4	BOOL	// Cage 18 bobbin 12 counter increase auxiliary
"M74.5"	M 74.5	BOOL	// Aux. M74.6
"M74.6"	M 74.6	BOOL	// Cage 18 bobbin 13 wire break on
"M74.7"	M 74.7	BOOL	// Cage 18 bobbin 13 counter increase auxiliary
"M75.0"	M 75.0	BOOL	// Aux. M75.1
"M75.1"	M 75.1	BOOL	// Cage 18 bobbin 14 wire break on
"M75.2"	M 75.2	BOOL	// Cage 18 bobbin 14 counter increase auxiliary
"M75.3"	M 75.3	BOOL	// Aux. M75.4
"M75.4"	M 75.4	BOOL	// Cage 18 bobbin 15 wire break on
"M75.5"	M 75.5	BOOL	// Cage 18 bobbin 15 counter increase auxiliary
"M75.6"	M 75.6	BOOL	// Aux. M75.7
"M75.7"	M 75.7	BOOL	// Cage 18 bobbin 16 wire break on
"M76.0"	M 76.0	BOOL	// Cage 18 bobbin 16 counter increase auxiliary
"M76.1"	M 76.1	BOOL	// Aux. M76.2
"M76.2"	M 76.2	BOOL	// Cage 18 bobbin 17 wire break on
"M76.3"	M 76.3	BOOL	// Cage 18 bobbin 17 counter increase auxiliary
"M76.4"	M 76.4	BOOL	// Aux. M76.5
"M76.5"	M 76.5	BOOL	// Cage 18 bobbin 18 wire break on
"M80.0"	M 80.0	BOOL	// Cage 24 bobbins wire break control insertion
"M80.1"	M 80.1	BOOL	// Aux. M80.2
"M80.2"	M 80.2	BOOL	// Cage 24 bobbin 1 wire break on
"M80.3"	M 80.3	BOOL	// Cage 24 bobbin 1 counter increase auxiliary
"M80.4"	M 80.4	BOOL	// Aux. M80.5
"M80.5"	M 80.5	BOOL	// Cage 24 bobbin 2 wire break on
"M80.6"	M 80.6	BOOL	// Cage 24 bobbin 2 counter increase auxiliary
"M80.7"	M 80.7	BOOL	// Aux. M81.7
"M81.0"	M 81.0	BOOL	// Cage 24 bobbin 3 wire break on
"M81.1"	M 81.1	BOOL	// Cage 24 bobbin 3 counter increase auxiliary
"M81.2"	M 81.2	BOOL	// Aux. M81.3
"M81.3"	M 81.3	BOOL	// Cage 24 bobbin 4 wire break on
"M81.4"	M 81.4	BOOL	// Cage 24 bobbin 4 counter increase auxiliary
"M81.5"	M 81.5	BOOL	// Aux. M81.6
"M81.6"	M 81.6	BOOL	// Cage 24 bobbin 5 wire break on
"M81.7"	M 81.7	BOOL	// Cage 24 bobbin 5 counter increase auxiliary
"M82.0"	M 82.0	BOOL	// Aux. M82.1
"M82.1"	M 82.1	BOOL	// Cage 24 bobbin 6 wire break on
"M82.2"	M 82.2	BOOL	// Cage 24 bobbin 6 counter increase auxiliary
"M82.3"	M 82.3	BOOL	// Aux. M82.4
"M82.4"	M 82.4	BOOL	// Cage 24 bobbin 7 wire break on
"M82.5"	M 82.5	BOOL	// Cage 24 bobbin 7 counter increase auxiliary
"M82.6"	M 82.6	BOOL	// Aux. M82.7
"M82.7"	M 82.7	BOOL	// Cage 24 bobbin 8 wire break on
"M83.1"	M 83.1	BOOL	// Aux. M83.2
"M83.2"	M 83.2	BOOL	// Cage 24 bobbin 9 wire break on
"M83.3"	M 83.3	BOOL	// Cage 24 bobbin 9 counter increase auxiliary
"M83.4"	M 83.4	BOOL	// Aux. M83.5
"M83.5"	M 83.5	BOOL	// Cage 24 bobbin 10 wire break on
"M83.6"	M 83.6	BOOL	// Cage 24 bobbin 10 counter increase auxiliary
"M83.7"	M 83.7	BOOL	// Aux. M84.0
"M84.0"	M 84.0	BOOL	// Cage 24 bobbin 11 wire break on
"M84.1"	M 84.1	BOOL	// Cage 24 bobbin 11 counter increase auxiliary
"M84.2"	M 84.2	BOOL	// Aux. M84.3
"M84.3"	M 84.3	BOOL	// Cage 24 bobbin 12 wire break on
"M84.4"	M 84.4	BOOL	// Cage 24 bobbin 12 counter increase auxiliary
"M84.5"	M 84.5	BOOL	// Aux. M84.6
"M84.6"	M 84.6	BOOL	// Cage 24 bobbin 13 wire break on
"M84.7"	M 84.7	BOOL	// Cage 24 bobbin 13 counter increase auxiliary
"M85.0"	M 85.0	BOOL	// Aux. M85.1
"M85.1"	M 85.1	BOOL	// Cage 24 bobbin 14 wire break on
"M85.2"	M 85.2	BOOL	// Cage 24 bobbin 14 counter increase auxiliary
"M85.3"	M 85.3	BOOL	// Aux. M85.4
"M85.4"	M 85.4	BOOL	// Cage 24 bobbin 15 wire break on
"M85.5"	M 85.5	BOOL	// Cage 24 bobbin 15 counter increase auxiliary
"M85.6"	M 85.6	BOOL	// Aux. M85.7
"M85.7"	M 85.7	BOOL	// Cage 24 bobbin 16 wire break on
"M86.0"	M 86.0	BOOL	// Cage 24 bobbin 16 counter increase auxiliary
"M86.1"	M 86.1	BOOL	// Aux. M86.2
"M86.2"	M 86.2	BOOL	// Cage 24 bobbin 17 wire break on
"M86.3"	M 86.3	BOOL	// Cage 24 bobbin 17 counter increase auxiliary
"M86.4"	M 86.4	BOOL	// Aux. M86.5
"M86.5"	M 86.5	BOOL	// Cage 24 bobbin 18 wire break on
"M86.6"	M 86.6	BOOL	// Cage 24 bobbin 18 counter increase auxiliary
"M86.7"	M 86.7	BOOL	// Aux. M87.0
"M87.0"	M 87.0	BOOL	// Cage 24 bobbin 19 wire break on
"M87.1"	M 87.1	BOOL	// Cage 24 bobbin 19 counter increase auxiliary
"M87.2"	M 87.2	BOOL	// Aux. M87.3
"M87.3"	M 87.3	BOOL	// Cage 24 bobbin 20 wire break on
"M87.4"	M 87.4	BOOL	// Cage 24 bobbin 20 counter increase auxiliary
"M87.5"	M 87.5	BOOL	// Aux. M87.6
"M87.6"	M 87.6	BOOL	// Cage 24 bobbin 21 wire break on
"M87.7"	M 87.7	BOOL	// Cage 24 bobbin 21 counter increase auxiliary
"M88.0"	M 88.0	BOOL	// Aux. M88.1
"M88.1"	M 88.1	BOOL	// Cage 24 bobbin 22 wire break on
"M88.2"	M 88.2	BOOL	// Cage 24 bobbin 22 counter increase auxiliary
"M88.3"	M 88.3	BOOL	// Aux. M88.4
"M88.4"	M 88.4	BOOL	// Cage 24 bobbin 23 wire break on
"M88.5"	M 88.5	BOOL	// Cage 24 bobbin 23 counter increase auxiliary
"M88.6"	M 88.6	BOOL	// Aux. M88.7
"M88.7"	M 88.7	BOOL	// Cage 24 bobbin 24 wire break on
"M89.0"	M 89.0	BOOL	// Cage 24 bobbin 24 counter increase auxiliary
"M100.0"	M 100.0	BOOL	// Bobbin diameters calculation clock
"M102.0"	M 102.0	BOOL	// Run consent without take-up on
"M102.1"	M 102.1	BOOL	// Run consent with take-up on
"M120.0"	M 120.0	BOOL	// Cage 6 normal stop
"M120.1"	M 120.1	BOOL	// Cage 6 quick stop
"M120.2"	M 120.2	BOOL	// Cage 6 emergency stop
"M130.0"	M 130.0	BOOL	// Cage 12 normal stop
"M130.1"	M 130.1	BOOL	// Cage 12 quick stop
"M130.2"	M 130.2	BOOL	// Cage 12 emergency stop
"M140.0"	M 140.0	BOOL	// Cage 18 normal stop
"M140.1"	M 140.1	BOOL	// Cage 18 quick stop
"M140.2"	M 140.2	BOOL	// Cage 18 emergency stop
"M150.0"	M 150.0	BOOL	// Cage 24 normal stop
"M150.1"	M 150.1	BOOL	// Cage 24 quick stop
"M150.2"	M 150.2	BOOL	// Cage 24 emergency stop
"M170.0"	M 170.0	BOOL	// Db100.dbx106.0 auxiliary
"M170.1"	M 170.1	BOOL	// Db100.dbx109.3 auxiliary
"M170.2"	M 170.2	BOOL	// Db100.dbx112.5 auxiliary
"M170.3"	M 170.3	BOOL	// Db100.dbx112.7 auxiliary
"M170.4"	M 170.4	BOOL	// Db100.dbx118.2 auxiliary
"M170.5"	M 170.5	BOOL	// Db100.dbx118.3 auxiliary
"M170.6"	M 170.6	BOOL	// Db100.dbx118.4 auxiliary
"M170.7"	M 170.7	BOOL	// Db100.dbx128.5 auxiliary
"M171.0"	M 171.0	BOOL	// Db100.dbx128.7 auxiliary
"M171.1"	M 171.1	BOOL	// Db100.dbx134.2 auxiliary
"M171.2"	M 171.2	BOOL	// Db100.dbx134.3 auxiliary
"M171.3"	M 171.3	BOOL	// Db100.dbx134.4 auxiliary
"M171.4"	M 171.4	BOOL	// Db100.dbx112.0 auxiliary
"M171.5"	M 171.5	BOOL	// Db100.dbx136.7 auxiliary
"M171.6"	M 171.6	BOOL	// Db100.dbx142.2 auxiliary
"M171.7"	M 171.7	BOOL	// Db100.dbx142.3 auxiliary
"M172.0"	M 172.0	BOOL	// Db100.dbx142.4 auxiliary
"M172.1"	M 172.1	BOOL	// Db100.dbx113.7 auxiliary
"M172.2"	M 172.2	BOOL	// Db100.dbx118.0 auxiliary
"M172.3"	M 172.3	BOOL	// Db100.dbx134.0 auxiliary
"M172.4"	M 172.4	BOOL	// Db100.dbx142.0 auxiliary
"M172.5"	M 172.5	BOOL	// Db100.dbx129.7 auxiliary
"M172.7"	M 172.7	BOOL	// Db100.dbx137.7 auxiliary
"M173.0"	M 173.0	BOOL	// Db100.dbx128.0 auxiliary
"M173.1"	M 173.1	BOOL	// Db100.dbx136.0 auxiliary
"M173.2"	M 173.2	BOOL	// Db100.dbx136.5 auxiliary
"M173.3"	M 173.3	BOOL	// Db100.dbx120.7 auxiliary
"M173.4"	M 173.4	BOOL	// DB100.DBX120.0 Auxliary
"M173.5"	M 173.5	BOOL	// Db100.dbx120.5 auxiliary
"M173.6"	M 173.6	BOOL	// Db100.dbx121.7 auxiliary
"M173.7"	M 173.7	BOOL	// Db100.dbx126.0 auxiliary
"M174.0"	M 174.0	BOOL	// Db100.dbx126.2 auxiliary
"M174.1"	M 174.1	BOOL	// Db100.dbx126.3 auxiliary
"M174.2"	M 174.2	BOOL	// Db100.dbx126.4 auxiliary
"M174.3"	M 174.3	BOOL	// Db100.dbx119.6 auxiliary
"M174.4"	M 174.4	BOOL	// Db100.dbx127.6 auxiliary
"M174.5"	M 174.5	BOOL	// Db100.dbx135.6 auxiliary
"M174.6"	M 174.6	BOOL	// Db100.dbx143.6 auxiliary
"M175.2"	M 175.2	BOOL	// DB100.DBX147.0 auxliary
"M175.3"	M 175.3	BOOL	// DB100.DBX147.1 auxliary
"M175.4"	M 175.4	BOOL	// DB100.DBX147.2 Auxliary
"M175.5"	M 175.5	BOOL	// DB100.dbx147.3 Auxliary
"M178.0"	M 178.0	BOOL	// Line run request
"M178.5"	M 178.5	BOOL	// Cage 6 wires break general alarm
"M178.6"	M 178.6	BOOL	// Cage 12 wires break general alarm
"M178.7"	M 178.7	BOOL	// Cage 18 wires break general alarm
"M179.0"	M 179.0	BOOL	// Cage 24 wires break general alarm
"M179.1"	M 179.1	BOOL	// Quick stop
"M179.2"	M 179.2	BOOL	// Cage 6 open pintles
"M179.3"	M 179.3	BOOL	// Cage 12 open pintles
"M179.4"	M 179.4	BOOL	// Cage 18 open pintles
"M179.5"	M 179.5	BOOL	// Cage 24 open pintles
"M179.6"	M 179.6	BOOL	// Linear speed calculation enable
"M180.0"	M 180.0	BOOL	// Line run without zero speed
"M180.1"	M 180.1	BOOL	// Line run with zero speed
"M180.3"	M 180.3	BOOL	// Line jog
"M180.4"	M 180.4	BOOL	// Loading run from cage 6 with piston disengaged
"M180.5"	M 180.5	BOOL	// Loading run from cage 12 with piston disengaged
"M180.6"	M 180.6	BOOL	// Loading run from cage 18 with piston disengaged
"M180.7"	M 180.7	BOOL	// Loading run from cage 24 with piston disengaged
"M181.2"	M 181.2	BOOL	// Loading run from cage 6
"M181.3"	M 181.3	BOOL	// Loading run from cage 12
"M181.4"	M 181.4	BOOL	// Loading run from cage 18
"M181.5"	M 181.5	BOOL	// Loading run from cage 24
"M182.0"	M 182.0	BOOL	// Take-up traverse run
"M182.1"	M 182.1	BOOL	// Take-up traverse left quick jog
"M182.2"	M 182.2	BOOL	// Take-up traverse right quick jog
"M182.3"	M 182.3	BOOL	// Take-up traverse positive home positioning
"M182.4"	M 182.4	BOOL	// Take-up traverse negative home positioning
"M182.5"	M 182.5	BOOL	// Take-up traverse home positioning run
"M183.0"	M 183.0	BOOL	// Take-up bobbin run
"M183.1"	M 183.1	BOOL	// Take-up bobbin forward jog
"M183.2"	M 183.2	BOOL	// Take-up bobbin backward jog
"M183.3"	M 183.3	BOOL	// Take-up bobbin run with zero speed
"M183.4"	M 183.4	BOOL	// Take-up bobbin jog with zero speed
"M184.0"	M 184.0	BOOL	// Capstan forward jog
"M184.1"	M 184.1	BOOL	// Capstan backward jog
"M184.2"	M 184.2	BOOL	// Capstan jog with zero speed
"M186.0"	M 186.0	BOOL	// Cage 18 on
"M186.1"	M 186.1	BOOL	// First loading run from cage 18
"M186.2"	M 186.2	BOOL	// Cage 18 z rotation
"M186.3"	M 186.3	BOOL	// Cage 18 s rotation
"M186.4"	M 186.4	BOOL	// Cage 18 ac motor jog for loading stroke
"M186.5"	M 186.5	BOOL	// Cage 18 loading protections
"M187.3"	M 187.3	BOOL	// Cage 18 preforming on
"M187.4"	M 187.4	BOOL	// Cage 18 preforming Z rotation selection
"M187.5"	M 187.5	BOOL	// Cage 18 preforming S rotation selection
"M188.0"	M 188.0	BOOL	// Cage 12 on
"M188.1"	M 188.1	BOOL	// First loading run from cage 12
"M188.2"	M 188.2	BOOL	// Cage 12 z rotation
"M188.3"	M 188.3	BOOL	// Cage 12 s rotation
"M188.4"	M 188.4	BOOL	// Cage 12 ac motor jog for loading stroke
"M188.5"	M 188.5	BOOL	// Cage 12 loading protections
"M189.3"	M 189.3	BOOL	// Cage 12 preforming on
"M189.4"	M 189.4	BOOL	// Cage 12 preforming Z rotation selection
"M189.5"	M 189.5	BOOL	// Cage 12 preforming S rotation selection
"M190.0"	M 190.0	BOOL	// Cage 6 on
"M190.1"	M 190.1	BOOL	// First loading run from cage 6
"M190.2"	M 190.2	BOOL	// Cage 6 z rotation
"M190.3"	M 190.3	BOOL	// Cage 6 s rotation
"M190.4"	M 190.4	BOOL	// Cage 6 ac motor jog for loading stroke
"M190.5"	M 190.5	BOOL	// Cage 6 loading protections
"M192.0"	M 192.0	BOOL	// Cage 24 on
"M192.1"	M 192.1	BOOL	// First loading run from Cage 24
"M192.2"	M 192.2	BOOL	// Cage 24 z rotation
"M192.3"	M 192.3	BOOL	// Cage 24 s rotation
"M192.4"	M 192.4	BOOL	// Cage 24 ac motor jog for loading stroke
"M192.5"	M 192.5	BOOL	// Cage 24 loading protections
"M193.3"	M 193.3	BOOL	// Cage 24 preforming on
"M193.4"	M 193.4	BOOL	// Cage 24 preforming Z rotation selection
"M193.5"	M 193.5	BOOL	// Cage 24 preforming S rotation selection
"M195.0"	M 195.0	BOOL	// Take-up traverse general alarm
"M195.1"	M 195.1	BOOL	// Take-up general alarm
"M195.3"	M 195.3	BOOL	// Cage 24 general alarm
"M195.4"	M 195.4	BOOL	// Cage 24 preforming general alarm
"M195.5"	M 195.5	BOOL	// Cage 18 general alarm
"M195.6"	M 195.6	BOOL	// Cage 18 preforming general alarm
"M195.7"	M 195.7	BOOL	// Cage 12 general alarm
"M196.0"	M 196.0	BOOL	// Cage 12 preforming general alarm
"M196.1"	M 196.1	BOOL	// Cage 6 general alarm
"M196.2"	M 196.2	BOOL	// Cage 6 preforming general alarm
"M196.3"	M 196.3	BOOL	// Pay-off 630 general alarm
"M196.7"	M 196.7	BOOL	// Metercounter general alarm
"M197.0"	M 197.0	BOOL	// Line general alarm
"M197.3"	M 197.3	BOOL	// Capstan general alarm
"M200.1"	M 200.1	BOOL	// Material from HMI (0=copper; 1=alluminium)
"M200.2"	M 200.2	BOOL	// Straight sectoral production
"M200.3"	M 200.3	BOOL	// Preformed sectoral production
"M200.4"	M 200.4	BOOL	// Round cable production
"M200.7"	M 200.7	BOOL	// Fixed ramp
"M201.0"	M 201.0	BOOL	// Bobbins diameters culculation set point
"M201.1"	M 201.1	BOOL	// Ramp enable
"M201.2"	M 201.2	BOOL	// Breaking control set point
"M202.0"	M 202.0	BOOL	// Cage 6 master of missing supply ramp down
"M202.1"	M 202.1	BOOL	// Cage 12 master of missing supply ramp down
"M202.2"	M 202.2	BOOL	// Cage 18 master of missing supply ramp down
"M202.3"	M 202.3	BOOL	// Cage 24 master of missing supply ramp down
"M220.0"	M 220.0	BOOL	// Missing power supply start
"M300.5"	M 300.5	BOOL	// FB125 All DP slaves ok
"MB304"	MB 304	BYTE	// FB125 slave adr
"ActualStep12"	MD 110	REAL	// Реальный шаг на 12-й клети
"ActualStep6"	MD 114	REAL	// Реальный шаг 6-й клети
"ActualStep18"	MD 121	REAL	// Реальный шаг 18-й клети
"ActualStep24"	MD 125	REAL	// Реальный шаг 24-й клети
"MD170"	MD 170	DWORD	// Auxiliary memory for alarms
"MD174"	MD 174	DWORD	// Auxiliary memory for alarms
"MW230"	MW 230	S5TIME	// T40 auxiliary
"MW232"	MW 232	S5TIME	// T42 auxiliary
"MW234"	MW 234	S5TIME	// T43 auxiliary
"MW236"	MW 236	S5TIME	// T44 auxiliary
"MW238"	MW 238	S5TIME	// T30 auxiliary
"MW240"	MW 240	S5TIME	// T32 auxiliary
"MW242"	MW 242	S5TIME	// T33 auxiliary
"MW244"	MW 244	S5TIME	// T25 auxiliary
"MW246"	MW 246	S5TIME	// T14 auxiliary
"MW248"	MW 248	S5TIME	// T16 auxiliary
"MW250"	MW 250	S5TIME	// T17 auxiliary
"MW252"	MW 252	S5TIME	// T18 auxiliary
"MW264"	MW 264	S5TIME	// T1 auxiliary
"MW266"	MW 266	S5TIME	// T2 auxiliary
"MW268"	MW 268	S5TIME	// T4 auxiliary
"M270"	MW 270	WORD	// T3 auxiliary
"MW272"	MW 272	WORD	// T20 auxiliary
"MW274"	MW 274	S5TIME	// T22 auxiliary
"MW276"	MW 276	S5TIME	// T23 auxiliary
"MW278"	MW 278	S5TIME	// T24 auxiliary
"MW284"	MW 284	WORD	// Cage 24 KIB activation point
"MW286"	MW 286	WORD	// Cage 24 KIB blocked/enabled
"MW288"	MW 288	WORD	// Cage 18 KIB activation point
"MW290"	MW 290	WORD	// Cage 12 activation point
"MW292"	MW 292	WORD	// Cage 6 activation point
"MW294"	MW 294	WORD	// Cage 18 KIB blocked/enabled
"MW296"	MW 296	WORD	// Cage 12 KIB blocked/enabled
"MW298"	MW 298	WORD	// Cage 6 KIB blocked/enabled
"Cycle execution"	OB 1	OB 1	// Cycle execution organization block
"Diagnostic interrupt"	OB 82	OB 82	// Diagnostic interrupt organization block
"Rack failure"	OB 86	OB 86	// Rack failure organization block
"Startup"	OB 100	OB 100	// Startup organization block
"MOD_ERR"	OB 122	OB 122	// Module Access Error
"PEB43"	PIB 43	BYTE	// Cage 24 peripheral input
"PEB53"	PIB 53	BYTE	// Cage 18 peripheral input
"PEB63"	PIB 63	BYTE	// Cage 12 peripheral input
"PEB73"	PIB 73	BYTE	// Cage 6 peripheral input
"PED260"	PID 260	DWORD	// Capstan motor encoder
"PED272"	PID 272	DWORD	// Take-up traverse encoder
"PED276"	PID 276	DWORD	// Take-up traverse count 24V/100kHz auxiliary
"PAD272"	PQD 272	DWORD	// Take-up traverse count 24V/100kHz enable
"PAW276"	PQW 276	WORD	// Take-up traverse count 24V/100kHz enable 1
"-659Y1"	PQW 278	WORD	// Cage 24 brake proportional valve
"-659Y2"	PQW 280	WORD	// Cage 24 bobbins brake proportional valve
"-559Y1"	PQW 282	WORD	// Cage 18 brake proportional valve
"-559Y2"	PQW 284	WORD	// Cage 18 bobbins brake proportional valve
"PAW286"	PQW 286	WORD	// Cage 12 brake proportional valve
"PAW288"	PQW 288	WORD	// Cage 12 bobbins brake proportional valve
"-359Y1"	PQW 290	WORD	// Cage 6 brake proportional valve
"-359Y2"	PQW 292	WORD	// Cage 6 bobbins brake proportional valve
"-359Y4"	PQW 296	WORD	// Pay-off 630 brake proportional valve
"-140G1:X101:9"	Q 0.0	BOOL	// Drives feeder start
"-922S3:LAMP"	Q 0.1	BOOL	// Take-up traverse quick left pilot lamp
"-922S4:LAMP"	Q 0.2	BOOL	// Take-up traverse quick right pilot lamp
"-925K3"	Q 0.3	BOOL	// Take-up bobbin run pilot lamps
"-732K1"	Q 0.4	BOOL	// Capstan motor blower contactor
"-732Y2"	Q 0.5	BOOL	// Capstan motor block brake electric valve
"-732Y3"	Q 0.6	BOOL	// Cable block opening electric valve
"-532K1"	Q 0.7	BOOL	// Cage 18 preforming motor electric brake relay
"-532K2"	Q 1.0	BOOL	// Cage 18 preforming motor blower contactor
"-532K3"	Q 1.1	BOOL	// Cage 18 motor blower contactor
"-532K4"	Q 1.2	BOOL	// Cage 18 loading motor s rotation contactor
"-532K5"	Q 1.3	BOOL	// Cage 18 loading motor z rotation contactor
"A001.4"	Q 1.4	BOOL	// Spare
"-532K7"	Q 1.5	BOOL	// Cage 18 guard blower motor contactor
"-432K1"	Q 1.6	BOOL	// Cage 12 preforming motor electric brake relay
"-432K2"	Q 1.7	BOOL	// Cage 12 preforming motor blower contactor
"-432K3"	Q 2.0	BOOL	// Cage 12 motor blower contactor
"-432K4"	Q 2.1	BOOL	// Cage 12 loading motor s rotation contactor
"-432K5"	Q 2.2	BOOL	// Cage 12 loading motor z rotation contactor
"A002.3"	Q 2.3	BOOL	// Spare
"-432K7"	Q 2.4	BOOL	// Cage 12 guard blower motor contactor
"-332K1"	Q 2.5	BOOL	// Cage 6 motor blower contactor
"-332K2"	Q 2.6	BOOL	// Cage 6 loading motor s rotation contactor
"-332K3"	Q 2.7	BOOL	// Cage 6 loading motor z rotation contactor
"A003.0"	Q 3.0	BOOL	// Spare
"-332K5"	Q 3.1	BOOL	// Cage 6 guard blower motor contactor
"-177S2:LAMP"	Q 3.2	BOOL	// Line run pilot lamp
"-183K2"	Q 3.3	BOOL	// Alarms reset pilot lamps
"-177S5:LAMP"	Q 3.4	BOOL	// Hold line speed pilot lamp
"-183K4"	Q 3.5	BOOL	// Line start siren
"-140G1:X101:10"	Q 3.6	BOOL	// Drives feeder reset
"-141A1:1"	Q 3.7	BOOL	// Breaking unit reset
"-632K1"	Q 4.0	BOOL	// Cage 24 preforming motor electric brake relay
"-632K2"	Q 4.1	BOOL	// Cage 24 preforming motor blower contactor
"-632K3"	Q 4.2	BOOL	// Cage 24 motor blower contactor
"-632K4"	Q 4.3	BOOL	// Cage 24 loading motor S rotation contactor
"-632K5"	Q 4.4	BOOL	// Cage 24 loading motor Z rotation contactor
"A004.5"	Q 4.5	BOOL	// Spare
"-632K7"	Q 4.6	BOOL	// Cage 24 guard  blower motor contactor
"A004.7"	Q 4.7	BOOL	// Spare
"-193K1"	Q 5.0	BOOL	// 230 VAC UPS automatic shut-down
"A005.1"	Q 5.1	BOOL	// Spare
"A005.2"	Q 5.2	BOOL	// Spare
"A005.3"	Q 5.3	BOOL	// Spare
"A005.4"	Q 5.4	BOOL	// Spare
"A005.5"	Q 5.5	BOOL	// Spare
"A005.6"	Q 5.6	BOOL	// Spare
"A005.7"	Q 5.7	BOOL	// Spare
"-MCB06:11"	Q 6.0	BOOL	// Cage 6 loader enable
"-MCB06:12"	Q 6.1	BOOL	// Cage 6 presence of bobbin inside cage
"-MCB06:13"	Q 6.2	BOOL	// Cage 6 loader lock piston inserted
"-MCB06:14"	Q 6.3	BOOL	// Cage 6 pintle open
"-MCB12:11"	Q 6.4	BOOL	// Cage 12 loader enable
"-MCB12:12"	Q 6.5	BOOL	// Cage 12 presence of bobbin inside cage
"-MCB12:13"	Q 6.6	BOOL	// Cage 12 loader lock piston inserted
"-MCB12:14"	Q 6.7	BOOL	// Cage 12 pintle open
"-MCB18:11"	Q 7.0	BOOL	// Cage 18 loader enable
"-MCB18:12"	Q 7.1	BOOL	// Cage 18 presence of bobbin inside cage
"-MCB18:13"	Q 7.2	BOOL	// Cage 18 loader lock piston inserted
"-MCB18:14"	Q 7.3	BOOL	// Cage 18 pintle open
"-MCB24:11"	Q 7.4	BOOL	// Cage 24 loader enable
"-MCB24:12"	Q 7.5	BOOL	// Cage 24 presence of bobbin inside cage
"-MCB24:13"	Q 7.6	BOOL	// Cage 24 loader lock piston inserted
"-MCB24:14"	Q 7.7	BOOL	// Cage 24 pintle open
"-981K1"	Q 32.0	BOOL	// Take-up idle pintle up motor contactor
"-981K2"	Q 32.1	BOOL	// Take-up idle pintle down motor contactor
"-981K3"	Q 32.2	BOOL	// Take-up driven pintle up motor contactor
"-981K4"	Q 32.3	BOOL	// Take-up driven pintle down motor contactor
"-981K5"	Q 33.0	BOOL	// Take-up idle pintle opening motor contactor
"-981K6"	Q 33.1	BOOL	// Take-up idle pintle closing motor contactor
"-981K7"	Q 33.2	BOOL	// Take-up traverse left direction pilot lamps
"-981K8"	Q 33.3	BOOL	// Take-up traverse right direction pilot lamps
"-982K1"	Q 34.0	BOOL	// Take-up traverse motor blower contactor
"-982K2"	Q 34.1	BOOL	// Take-up bobbin motor blower contactor
"-982K3"	Q 34.2	BOOL	// Take-up bobbin electric brake relay
"A034.3"	Q 34.3	BOOL	// Spare
"-682Y1"	Q 42.0	BOOL	// Cage 24 loading motor engaging electric valve
"-682Y2"	Q 42.1	BOOL	// Cage 24 loading motor disingaging electric valve
"-682Y3"	Q 42.2	BOOL	// Cage 24 cage block brake electric valve
"-683Y1"	Q 42.3	BOOL	// Cage 24 open air in cage electric valve
"-683Y2"	Q 42.4	BOOL	// Cage 24 close air in cage electric valve
"-683Y3"	Q 42.5	BOOL	// Cage 24 loading pinston engaging into cage electric valve
"-683Y4"	Q 42.6	BOOL	// Cage 24 loading pinston disengaging into cage electric valve
"-684Y5"	Q 42.7	BOOL	// Cage 24 pintles locking system opening electric valve
"-684Y6"	Q 43.0	BOOL	// Cage 24 pintles locking system closing electric valve
"-684Y7"	Q 43.1	BOOL	// Cage 24 pintles opening electric valve
"-684Y8"	Q 43.2	BOOL	// Cage 24 pintles closing electric valve
"-686Y1:LOCK"	Q 43.3	BOOL	// Cage 24 front door locking
"-684Y3"	Q 43.4	BOOL	// Cage 24 guard opening electric valve
"-684Y4"	Q 43.5	BOOL	// Cage 24 guard closing electric valve
"-663S3:LAMP"	Q 43.6	BOOL	// Cage 24 loading run pilot lamp
"-663S7:LAMP"	Q 43.7	BOOL	// Cage 24 loading insertion pilot lamp
"-687H1:LAMP"	Q 44.0	BOOL	// Cage 24 pintles open pilot lamp
"-687H2:LAMP"	Q 44.1	BOOL	// Cage 24 broken wire pilot lamp
"A044.2"	Q 44.2	BOOL	// Spare
"A044.3"	Q 44.3	BOOL	// Spare
"-663S4:LAMP"	Q 44.4	BOOL	// Cage 24 alarm reset pilot lamp
"-688Y1"	Q 44.5	BOOL	// Cage 24 loader lock piston valve
"-688Y2"	Q 44.6	BOOL	// Cage 24 loader unlock piston valve
"A044.7"	Q 44.7	BOOL	// Spare
"A045.0"	Q 45.0	BOOL	// Spare
"A045.1"	Q 45.1	BOOL	// Spare
"A045.2"	Q 45.2	BOOL	// Spare
"A045.3"	Q 45.3	BOOL	// Spare
"-688Y8:LOCK"	Q 45.4	BOOL	// Cage 24 preforming guard locking
"A045.5"	Q 45.5	BOOL	// Spare
"A045.6"	Q 45.6	BOOL	// Spare
"A045.7"	Q 45.7	BOOL	// Spare
"-582Y1"	Q 52.0	BOOL	// Cage 18 loading motor engaging electric valve
"-582Y2"	Q 52.1	BOOL	// Cage 18 loading motor disengaging electric valve
"-582Y3"	Q 52.2	BOOL	// Cage 18 block brake electric valve
"-583Y1"	Q 52.3	BOOL	// Cage 18 air inlet electric valve
"-583Y2"	Q 52.4	BOOL	// Cage 18 air outlet electric valve
"-583Y3"	Q 52.5	BOOL	// Cage 18 loading piston engaging into Cage electric valve
"-583Y4"	Q 52.6	BOOL	// Cage 18 loading piston disengaging from Cage electric valve
"-584Y5"	Q 52.7	BOOL	// Cage 18 pintles locking system opening electric valves
"-584Y6"	Q 53.0	BOOL	// Cage 18 pintles locking system closing electric valves
"-584Y7"	Q 53.1	BOOL	// Cage 18 pintles opening electric valves
"-584Y8"	Q 53.2	BOOL	// Cage 18 pintles closing electric valves
"-586Y1:LOCK"	Q 53.3	BOOL	// Cage 18 front door locking
"-586Y3"	Q 53.4	BOOL	// Cage 18 guard opening electric valve
"-586Y4"	Q 53.5	BOOL	// Cage 18 guard closing electric valve
"-563S3:LAMP"	Q 53.6	BOOL	// Cage 18 loading run pilot lamp
"-564S7:LAMP"	Q 53.7	BOOL	// Cage 18 loading insertion pilot lamp
"-587H1"	Q 54.0	BOOL	// Cage 18 pintles open pilot lamp
"-587H2"	Q 54.1	BOOL	// Cage 18 broken wire pilot lamp
"A054.2"	Q 54.2	BOOL	// Spare
"A054.3"	Q 54.3	BOOL	// Spare
"-563S4:LAMP"	Q 54.4	BOOL	// Cage 18 alarms reset pilot lamp
"-588Y1"	Q 54.5	BOOL	// Cage 18 loader unlock piston valve
"-588Y2"	Q 54.6	BOOL	// Cage 18 loader lock piston valve
"A054.7"	Q 54.7	BOOL	// Spare
"A055.0"	Q 55.0	BOOL	// Spare
"A055.1"	Q 55.1	BOOL	// Spare
"A055.2"	Q 55.2	BOOL	// Spare
"A055.3"	Q 55.3	BOOL	// Spare
"-565Y8:LOCK"	Q 55.4	BOOL	// Cage 18 preforming guard locking
"A055.5"	Q 55.5	BOOL	// Spare
"A055.6"	Q 55.6	BOOL	// Spare
"A055.7"	Q 55.7	BOOL	// Spare
"-482Y1"	Q 62.0	BOOL	// Cage 12 loading motor engaging electric valve
"-482Y2"	Q 62.1	BOOL	// Cage 12 loading motor disengaging electric valve
"-482Y3"	Q 62.2	BOOL	// Cage 12 block brake electric valve
"-483Y1"	Q 62.3	BOOL	// Cage 12 air inlet electric valve
"-483Y2"	Q 62.4	BOOL	// Cage 12 air outlet electric valve
"-483Y3"	Q 62.5	BOOL	// Cage 12 loading piston engaging into cage electric valve
"-483Y4"	Q 62.6	BOOL	// Cage 12 loading piston disengaging from cage electric valve
"-484Y5"	Q 62.7	BOOL	// Cage 12 pintles locking system opening electric valves
"-484Y6"	Q 63.0	BOOL	// Cage 12 pintles locking system closing electric valves
"-484Y7"	Q 63.1	BOOL	// Cage 12 pintles opening electric valves
"-484Y8"	Q 63.2	BOOL	// Cage 12 pintles closing electric valves
"-486Y1:LOCK"	Q 63.3	BOOL	// Cage 12 front door locking
"-486Y3"	Q 63.4	BOOL	// Cage 12 guard opening electric valve
"-486Y4"	Q 63.5	BOOL	// Cage 12 guard closing electric valve
"-463S3:LAMP"	Q 63.6	BOOL	// Cage 12 loading run pilot lamp
"-463S7:LAMP"	Q 63.7	BOOL	// Cage 12 loading insertion pilot lamp
"-487H1:LAMP"	Q 64.0	BOOL	// Cage 12 pintles open pilot lamp
"-487H2:LAMP"	Q 64.1	BOOL	// Cage 12 broken wire pilot lamp
"A064.2"	Q 64.2	BOOL	// Spare
"A064.3"	Q 64.3	BOOL	// Spare
"-463S4:LAMP"	Q 64.4	BOOL	// Cage 12 alarms reset pilot lamp
"-488Y1"	Q 64.5	BOOL	// Cage 12 loader unlock piston valve
"-488Y2"	Q 64.6	BOOL	// Cage 12 loader lock piston valve
"A064.7"	Q 64.7	BOOL	// Spare
"A065.0"	Q 65.0	BOOL	// Spare
"A065.1"	Q 65.1	BOOL	// Spare
"A065.2"	Q 65.2	BOOL	// Spare
"A065.3"	Q 65.3	BOOL	// Spare
"-489Y8:LOCK"	Q 65.4	BOOL	// Cage 12 preforming guard locking
"A065.5"	Q 65.5	BOOL	// Spare
"A065.6"	Q 65.6	BOOL	// Spare
"A065.7"	Q 65.7	BOOL	// Spare
"-382Y1"	Q 72.0	BOOL	// Cage 6 loading motor engaging electric valve
"-382Y2"	Q 72.1	BOOL	// Cage 6 loading motor disengaging electric valve
"-382Y3"	Q 72.2	BOOL	// Cage 6 block stationary brake electric valve
"-383Y1"	Q 72.3	BOOL	// Cage 6 air inlet electric valve
"-383Y2"	Q 72.4	BOOL	// Cage 6 air outlet electric valve
"-383Y3"	Q 72.5	BOOL	// Cage 6 loading piston engaging into cage electric valve
"-383Y4"	Q 72.6	BOOL	// Cage 6 loading piston disengaging from cage electric valve
"-384K1"	Q 72.7	BOOL	// Cage 6 pintles locking system opening electric valves
"-384K2"	Q 73.0	BOOL	// Cage 6 pintles locking system closing electric valves
"-384K3"	Q 73.1	BOOL	// Cage 6 pintles opening electric valves
"-384K4"	Q 73.2	BOOL	// Cage 6 pintles closing electric valves
"-386Y1:LOCK"	Q 73.3	BOOL	// Cage 6 front door locking
"-386Y3"	Q 73.4	BOOL	// Cage 6 guard opening electric valve
"-386Y4"	Q 73.5	BOOL	// Cage 6 guard closing electric valve
"-363S3:LAMP"	Q 73.6	BOOL	// Cage 6 loading run pilot lamp
"-364S7:LAMP"	Q 73.7	BOOL	// Cage 6 loading insertion pilot lamp
"-387H1:LAMP"	Q 74.0	BOOL	// Cage 6 pintles open pilot lamp
"-387H2:LAMP"	Q 74.1	BOOL	// Cage 6 broken wire pilot lamp
"A074.2"	Q 74.2	BOOL	// Spare
"A074.3"	Q 74.3	BOOL	// Spare
"-363S4:LAMP"	Q 74.4	BOOL	// Cage 6 alarms reset pilot lamp
"-388Y1"	Q 74.5	BOOL	// Cage 6 loader unlock piston valve
"-388Y2"	Q 74.6	BOOL	// Cage 6 loader lock piston valve
"A074.7"	Q 74.7	BOOL	// Spare
"A075.0"	Q 75.0	BOOL	// Spare
"A075.1"	Q 75.1	BOOL	// Spare
"A075.2"	Q 75.2	BOOL	// Spare
"A075.3"	Q 75.3	BOOL	// Spare
"-388Y8:LOCK"	Q 75.4	BOOL	// Cage 6 preforming guard locking
"-390H1:LAMP"	Q 75.5	BOOL	// Central Pay-off 630 broken wire pilot lamp
"-390H2:LAMP"	Q 75.6	BOOL	// Central Pay-off 630 pintle open pilot lamp
"-390K3"	Q 75.7	BOOL	// Central Pay-off 630 pintle enable
"GADR_LGC"	SFC 5	SFC 5	// Query logical address of a channel
"RD_SINFO"	SFC 6	SFC 6	// Read OB start information
"DPNRM_DG"	SFC 13	SFC 13	// Read diagnostic data of a DP slave
"DPRD_DAT"	SFC 14	SFC 14	// Read Consistent Data of a Standard DP Slave
"DPWR_DAT"	SFC 15	SFC 15	// Write Consistent Data to a Standard DP Slave
"DIS_AIRT"	SFC 41	SFC 41	// Delay the higher priority interrupts and asynchronous errors
"EN_AIRT"	SFC 42	SFC 42	// Enable higher priority interrupts and asynchronous errors
"LGC_GADR"	SFC 49	SFC 49	// Query the module slot belonging to a logical address
"RDSYSST"	SFC 51	SFC 51	// Read a system status list or partial list
"T0"	T 0	TIMER	// Auxiliary on on-delay timer
"T1"	T 1	TIMER	// Breaking control on-delay timer
"T2"	T 2	TIMER	// Brakes-oil control on-delay timer
"T3"	T 3	TIMER	// Guards blowers off-delay timer
"T4"	T 4	TIMER	// Line run on-delay timer
"T5"	T 5	TIMER	// Bobbin diameters calculation on-delay timer
"T6"	T 6	TIMER	// Ac motor drives feeder breaking resistor alarm control on-delay timer
"T10"	T 10	TIMER	// Take-up traverse motor drive off-delay timer
"T11"	T 11	TIMER	// Take-up driven pintle up on-delay timer
"T12"	T 12	TIMER	// Take-up idle pintle up on-delay timer
"T13"	T 13	TIMER	// Time Lock Door
"T14"	T 14	TIMER	// Cage 24 brakes block open on-delay timer
"T15"	T 15	TIMER	// Cage 24 motor jog extended pulse timer for loading stroke
"T16"	T 16	TIMER	// Cage 24 piston inside cage on-delay timer
"T17"	T 17	TIMER	// Cage 24 piston outside cage on-delay timer
"T18"	T 18	TIMER	// Cage 24 air inlet on-delay timer
"T19"	T 19	TIMER	// Cage 24 open front door control on-delay timer
"T20"	T 20	TIMER	// Cage 18 brakes block open on-delay timer
"T21"	T 21	TIMER	// Cage 18 motor jog extended pulse timer for loading stroke
"T22"	T 22	TIMER	// Cage 18 piston inside cage on-delay timer
"T23"	T 23	TIMER	// Cage 18 piston outside cage on-delay timer
"T24"	T 24	TIMER	// Cage 18 air inlet on-delay timer
"T25"	T 25	TIMER	// Cage 18 open front door control on-delay timer
"T30"	T 30	TIMER	// Cage 12 brakes block open on-delay timer
"T31"	T 31	TIMER	// Cage 12 motor jog extended pulse timer for loading stroke
"T32"	T 32	TIMER	// Cage 12 piston inside cage on-delay timer
"T33"	T 33	TIMER	// Cage 12 piston outside cage on-delay timer
"T34"	T 34	TIMER	// Cage 12 air inlet on-delay timer
"T35"	T 35	TIMER	// Cage 12 open front door control on-delay timer
"T40"	T 40	TIMER	// Cage 6 brakes block open on-delay timer
"T41"	T 41	TIMER	// Cage 6 motor jog extended pulse timer for loading stroke
"T42"	T 42	TIMER	// Cage 6 piston inside cage on-delay timer
"T43"	T 43	TIMER	// Cage 6 piston outside cage on-delay timer
"T44"	T 44	TIMER	// Cage 6 air inlet on-delay timer
"T45"	T 45	TIMER	// Cage 6 open front door control on-delay timer
"Dalarm_24"	T 50	TIMER	// Задержка на подсчет катушек
"Dalarm_18"	T 51	TIMER	// Задержка на подсчет катушек
"Dalarm_12"	T 52	TIMER	// Задержка на подсчет катушек
"Dalarm_6"	T 53	TIMER	// Задержка на подсчет катушек
"T100"	T 100	TIMER	// Cage 6 bobbin 1 wire break on-delay timer 1
"T101"	T 101	TIMER	// Cage 6 bobbin 2 wire break on-delay timer 1
"T102"	T 102	TIMER	// Cage 6 bobbin 3 wire break on-delay timer 1
"T103"	T 103	TIMER	// Cage 6 bobbin 4 wire break on-delay timer 1
"T104"	T 104	TIMER	// Cage 6 bobbin 5 wire break on-delay timer 1
"T105"	T 105	TIMER	// Cage 6 bobbin 6 wire break on-delay timer 1
"T106"	T 106	TIMER	// Cage 12 bobbin 1 wire break on-delay timer 1
"T107"	T 107	TIMER	// Cage 12 bobbin 2 wire break on-delay timer 1
"T108"	T 108	TIMER	// Cage 12 bobbin 3 wire break on-delay timer 1
"T109"	T 109	TIMER	// Cage 12 bobbin 4 wire break on-delay timer 1
"T110"	T 110	TIMER	// Cage 12 bobbin 5 wire break on-delay timer 1
"T111"	T 111	TIMER	// Cage 12 bobbin 6 wire break on-delay timer 1
"T112"	T 112	TIMER	// Cage 12 bobbin 7 wire break on-delay timer 1
"T113"	T 113	TIMER	// Cage 12 bobbin 8 wire break on-delay timer 1
"T114"	T 114	TIMER	// Cage 12 bobbin 9 wire break on-delay timer 1
"T115"	T 115	TIMER	// Cage 12 bobbin 10 wire break on-delay timer 1
"T116"	T 116	TIMER	// Cage 12 bobbin 11 wire break on-delay timer 1
"T117"	T 117	TIMER	// Cage 12 bobbin 12 wire break on-delay timer 1
"T118"	T 118	TIMER	// Cage 18 bobbin 1 wire break on-delay timer 1
"T119"	T 119	TIMER	// Cage 18 bobbin 2 wire break on-delay timer 1
"T120"	T 120	TIMER	// Cage 18 bobbin 3 wire break on-delay timer 1
"T121"	T 121	TIMER	// Cage 18 bobbin 4 wire break on-delay timer 1
"T122"	T 122	TIMER	// Cage 18 bobbin 5 wire break on-delay timer 1
"T123"	T 123	TIMER	// Cage 18 bobbin 6 wire break on-delay timer 1
"T124"	T 124	TIMER	// Cage 18 bobbin 7 wire break on-delay timer 1
"T125"	T 125	TIMER	// Cage 18 bobbin 8 wire break on-delay timer 1
"T126"	T 126	TIMER	// Cage 18 bobbin 9 wire break on-delay timer 1
"T127"	T 127	TIMER	// Cage 18 bobbin 10 wire break on-delay timer 1
"T128"	T 128	TIMER	// Cage 18 bobbin 11 wire break on-delay timer 1
"T129"	T 129	TIMER	// Cage 18 bobbin 12 wire break on-delay timer 1
"T130"	T 130	TIMER	// Cage 18 bobbin 13 wire break on-delay timer 1
"T131"	T 131	TIMER	// Cage 18 bobbin 14 wire break on-delay timer 1
"T132"	T 132	TIMER	// Cage 18 bobbin 15 wire break on-delay timer 1
"T133"	T 133	TIMER	// Cage 18 bobbin 16 wire break on-delay timer 1
"T134"	T 134	TIMER	// Cage 18 bobbin 17 wire break on-delay timer 1
"T135"	T 135	TIMER	// Cage 18 bobbin 18 wire break on-delay timer 1
"T136"	T 136	TIMER	// Cage 24 bobbin 1 wire break on-delay timer 1
"T137"	T 137	TIMER	// Cage 24 bobbin 2 wire break on-delay timer 1
"T138"	T 138	TIMER	// Cage 24 bobbin 3 wire break on-delay timer 1
"T139"	T 139	TIMER	// Cage 24 bobbin 4 wire break on-delay timer 1
"T140"	T 140	TIMER	// Cage 24 bobbin 5 wire break on-delay timer 1
"T141"	T 141	TIMER	// Cage 24 bobbin 6 wire break on-delay timer 1
"T142"	T 142	TIMER	// Cage 24 bobbin 7 wire break on-delay timer 1
"T143"	T 143	TIMER	// Cage 24 bobbin 8 wire break on-delay timer 1
"T144"	T 144	TIMER	// Cage 24 bobbin 9 wire break on-delay timer 1
"T145"	T 145	TIMER	// Cage 24 bobbin 10 wire break on-delay timer 1
"T146"	T 146	TIMER	// Cage 24 bobbin 11 wire break on-delay timer 1
"T147"	T 147	TIMER	// Cage 24 bobbin 12 wire break on-delay timer 1
"T148"	T 148	TIMER	// Cage 24 bobbin 13 wire break on-delay timer 1
"T149"	T 149	TIMER	// Cage 24 bobbin 14 wire break on-delay timer 1
"T150"	T 150	TIMER	// Cage 24 bobbin 15 wire break on-delay timer 1
"T151"	T 151	TIMER	// Cage 24 bobbin 16 wire break on-delay timer 1
"T152"	T 152	TIMER	// Cage 24 bobbin 17 wire break on-delay timer 1
"T153"	T 153	TIMER	// Cage 24 bobbin 18 wire break on-delay timer 1
"T154"	T 154	TIMER	// Cage 24 bobbin 19 wire break on-delay timer 1
"T155"	T 155	TIMER	// Cage 24 bobbin 20 wire break on-delay timer 1
"T156"	T 156	TIMER	// Cage 24 bobbin 21 wire break on-delay timer 1
"T157"	T 157	TIMER	// Cage 24 bobbin 22 wire break on-delay timer 1
"T158"	T 158	TIMER	// Cage 24 bobbin 23 wire break on-delay timer 1
"T159"	T 159	TIMER	// Cage 24 bobbin 24 wire break on-delay timer 1
"T160"	T 160	TIMER	// Pay-off 630 bobbin wire break on-delay timer
"VAT_1"	VAT 1	
"Kosta"	VAT 2	
"steps"	VAT 3	
END_SYMBOL_TABLE

// FB 125: know-how protected block, not included

FUNCTION "Alarms Reset" : VOID	// FC 1
TITLE = ALARMS RESET FUNCTION
AUTHOR : Milesi
VERSION : 0.1
BEGIN
NETWORK
TITLE = ALARMS RESET
      L     0;
      T     DB100.DBD 100;
      T     DB100.DBD 104;
      T     DB100.DBD 108;
      T     DB100.DBD 112;
      T     DB100.DBD 116;
      T     DB100.DBD 120;
      T     DB100.DBD 124;
      T     DB100.DBD 128;
      T     DB100.DBD 132;
      T     DB100.DBD 136;
      T     DB100.DBD 140;
      T     DB100.DBD 144;
      T     DB100.DBD 148;
      T     "MD170";
      T     "MD174";
END_FUNCTION

FUNCTION "Profibus alarms" : VOID	// FC 2
TITLE = PROFIBUS ALARMS FUNCTION
AUTHOR : Milesi
VERSION : 0.1
BEGIN
// (block stored without names or comments; labels and parameter names are numbered)
END_FUNCTION

FUNCTION "Profibus unit" : VOID	// FC 3
TITLE = PROFIBUS UNIT FUNCTION
AUTHOR : Milesi
VERSION : 0.1
BEGIN
NETWORK
TITLE = CAGE 24 WRITE PKW (P517)
//Dec 517 = Hex 205
      A     "M1.5";
      JC    J00;
      L     W#16#2205;
      T     "Plc --> Drives".PKW_WRITE_CAGE24.DB2_DBW500;
      L     0;
      T     "Plc --> Drives".PKW_WRITE_CAGE24.DB2_DBW502;
      L     "MW286";
      T     "Plc --> Drives".PKW_WRITE_CAGE24.DB2_DBW506;
J00:  NOP   0;
NETWORK
TITLE = CAGE 24 WRITE PKW (P518)
//Dec 518 = Hex 206
      A     "M1.5";
      JCN   J01;
      L     W#16#2206;
      T     "Plc --> Drives".PKW_WRITE_CAGE24.DB2_DBW500;
      L     0;
      T     "Plc --> Drives".PKW_WRITE_CAGE24.DB2_DBW502;
      L     "MW284";
      T     "Plc --> Drives".PKW_WRITE_CAGE24.DB2_DBW506;
J01:  NOP   0;
NETWORK
TITLE = READ/WRITE PKW FROM/TO DRIVE CAGE 24 (ADDRESS 7)
//Dec 390 = Hex 186
      CALL  "DPRD_DAT" (
           LADDR                    := W#16#186,
           RET_VAL                  := "Profibus SFC Alarm".DB3_DBW36,
           RECORD                   := "Drives --> Plc".PKW_READ_CAGE24);
      CALL  "DPWR_DAT" (
           LADDR                    := W#16#186,
           RECORD                   := "Plc --> Drives".PKW_WRITE_CAGE24,
           RET_VAL                  := "Profibus SFC Alarm".DB3_DBW38);
NETWORK
TITLE = CAGE 18 WRITE PKW (P517)
//Dec 517 = Hex 205
      A     "M1.5";
      JC    J02;
      L     W#16#2205;
      T     "Plc --> Drives".PKW_WRITE_CAGE18.DB2_DBW510;
      L     0;
      T     "Plc --> Drives".PKW_WRITE_CAGE18.DB2_DBW512;
      L     "MW294";
      T     "Plc --> Drives".PKW_WRITE_CAGE18.DB2_DBW516;
J02:  NOP   0;
NETWORK
TITLE = CAGE 18 WRITE PKW (P518)
//Dec 518 = Hex 206
      A     "M1.5";
      JCN   J03;
      L     W#16#2206;
      T     "Plc --> Drives".PKW_WRITE_CAGE18.DB2_DBW510;
      L     0;
      T     "Plc --> Drives".PKW_WRITE_CAGE18.DB2_DBW512;
      L     "MW288";
      T     "Plc --> Drives".PKW_WRITE_CAGE18.DB2_DBW516;
J03:  NOP   0;
NETWORK
TITLE = READ/WRITE PKW FROM/TO DRIVE CAGE 18 (ADDRESS 9)
//Dec 422 = Hex 1A6
      CALL  "DPRD_DAT" (
           LADDR                    := W#16#1A6,
           RET_VAL                  := "Profibus SFC Alarm".DB3_DBW16,
           RECORD                   := "Drives --> Plc".PKW_READ_CAGE18);
      CALL  "DPWR_DAT" (
           LADDR                    := W#16#1A6,
           RECORD                   := "Plc --> Drives".PKW_WRITE_CAGE18,
           RET_VAL                  := "Profibus SFC Alarm".DB3_DBW18);
NETWORK
TITLE = CAGE 12 WRITE PKW (P517)
//Dec 517 = Hex 205
      A     "M1.5";
      JC    J06;
      L     W#16#2205;
      T     "Plc --> Drives".PKW_WRITE_CAGE12.DB2_DBW520;
      L     0;
      T     "Plc --> Drives".PKW_WRITE_CAGE12.DB2_DBW522;
      L     "MW296";
      T     "Plc --> Drives".PKW_WRITE_CAGE12.DB2_DBW526;
J06:  NOP   0;
NETWORK
TITLE = CAGE 12 WRITE PKW (P518)
//Dec 518 = Hex 206
      A     "M1.5";
      JCN   J07;
      L     W#16#2206;
      T     "Plc --> Drives".PKW_WRITE_CAGE12.DB2_DBW520;
      L     0;
      T     "Plc --> Drives".PKW_WRITE_CAGE12.DB2_DBW522;
      L     "MW290";
      T     "Plc --> Drives".PKW_WRITE_CAGE12.DB2_DBW526;
J07:  NOP   0;
NETWORK
TITLE = READ/WRITE PKW FROM/TO DRIVE CAGE 12 (ADDRESS 11)
//Dec 438 = Hex 1B6
      CALL  "DPRD_DAT" (
           LADDR                    := W#16#B6,
           RET_VAL                  := "Profibus SFC Alarm".DB3_DBW24,
           RECORD                   := "Drives --> Plc".PKW_READ_CAGE12);
      CALL  "DPWR_DAT" (
           LADDR                    := W#16#1B6,
           RECORD                   := "Plc --> Drives".PKW_WRITE_CAGE12,
           RET_VAL                  := "Profibus SFC Alarm".DB3_DBW26);
NETWORK
TITLE = CAGE 6 WRITE PKW (P517)
//Dec 517 = Hex 205
      A     "M1.5";
      JC    J04;
      L     W#16#2205;
      T     "Plc --> Drives".PKW_WRITE_CAGE6.DB2_DBW530;
      L     0;
      T     "Plc --> Drives".PKW_WRITE_CAGE6.DB2_DBW532;
      L     "MW298";
      T     "Plc --> Drives".PKW_WRITE_CAGE6.DB2_DBW536;
J04:  NOP   0;
NETWORK
TITLE = CAGE 6 WRITE PKW (P518)
//Dec 518 = Hex 206
      A     "M1.5";
      JCN   J05;
      L     W#16#2206;
      T     "Plc --> Drives".PKW_WRITE_CAGE6.DB2_DBW530;
      L     0;
      T     "Plc --> Drives".PKW_WRITE_CAGE6.DB2_DBW532;
      L     "MW292";
      T     "Plc --> Drives".PKW_WRITE_CAGE6.DB2_DBW536;
J05:  NOP   0;
NETWORK
TITLE = READ/WRITE PKW FROM/TO DRIVE CAGE 6 (ADDRESS 12)
//Dec 446 = Hex 1BE
      CALL  "DPRD_DAT" (
           LADDR                    := W#16#1BE,
           RET_VAL                  := "Profibus SFC Alarm".DB3_DBW28,
           RECORD                   := "Drives --> Plc".PKW_READ_CAGE6);
      CALL  "DPWR_DAT" (
           LADDR                    := W#16#1BE,
           RECORD                   := "Plc --> Drives".PKW_WRITE_CAGE6,
           RET_VAL                  := "Profibus SFC Alarm".DB3_DBW30);
NETWORK
TITLE = READ/WRITE FROM/TO DRIVE TAKE-UP TRAVERSE (ADDRESS 3)
//Dec 400 = Hex 190
      CALL  "DPRD_DAT" (
           LADDR                    := W#16#190,
           RET_VAL                  := "Profibus SFC Alarm".DB3_DBW0,
           RECORD                   := P#DB1.DBX 0.0 BYTE 12);
      CALL  "DPWR_DAT" (
           LADDR                    := W#16#190,
           RECORD                   := P#DB2.DBX 0.0 BYTE 12,
           RET_VAL                  := "Profibus SFC Alarm".DB3_DBW2);
NETWORK
TITLE = READ/WRITE FROM/TO DRIVE TAKE-UP BOBBIN (ADDRESS 4)
//Dec 306 = Hex 132
      CALL  "DPRD_DAT" (
           LADDR                    := W#16#132,
           RET_VAL                  := "Profibus SFC Alarm".DB3_DBW4,
           RECORD                   := P#DB1.DBX 40.0 BYTE 12);
      CALL  "DPWR_DAT" (
           LADDR                    := W#16#132,
           RECORD                   := P#DB2.DBX 40.0 BYTE 12,
           RET_VAL                  := "Profibus SFC Alarm".DB3_DBW6);
NETWORK
TITLE = READ/WRITE FROM/TO DRIVE CAPSTAN (ADDRESS 5)
//Dec 318 = Hex 13E
      CALL  "DPRD_DAT" (
           LADDR                    := W#16#13E,
           RET_VAL                  := "Profibus SFC Alarm".DB3_DBW8,
           RECORD                   := P#DB1.DBX 80.0 BYTE 12);
      CALL  "DPWR_DAT" (
           LADDR                    := W#16#13E,
           RECORD                   := P#DB2.DBX 80.0 BYTE 12,
           RET_VAL                  := "Profibus SFC Alarm".DB3_DBW10);
NETWORK
TITLE = READ/WRITE FROM/TO DRIVE CAGE 24 FREFORMING (ADDRESS 6)
//Dec 466 = Hex 1D2
      CALL  "DPRD_DAT" (
           LADDR                    := W#16#1D2,
           RET_VAL                  := "Profibus SFC Alarm".DB3_DBW32,
           RECORD                   := P#DB1.DBX 120.0 BYTE 12);
      CALL  "DPWR_DAT" (
           LADDR                    := W#16#1D2,
           RECORD                   := P#DB2.DBX 120.0 BYTE 12,
           RET_VAL                  := "Profibus SFC Alarm".DB3_DBW34);
NETWORK
TITLE = READ/WRITE FROM/TO DRIVE CAGE 24 (ADDRESS 7)
//Dec 454 = Hex 1C6
      CALL  "DPRD_DAT" (
           LADDR                    := W#16#1C6,
           RET_VAL                  := "Profibus SFC Alarm".DB3_DBW48,
           RECORD                   := P#DB1.DBX 160.0 BYTE 12);
      CALL  "DPWR_DAT" (
           LADDR                    := W#16#1C6,
           RECORD                   := P#DB2.DBX 160.0 BYTE 12,
           RET_VAL                  := "Profibus SFC Alarm".DB3_DBW50);
NETWORK
TITLE = READ/WRITE FROM/TO DRIVE CAGE 18 FREFORMING (ADDRESS 8)
//Dec 330 = Hex 14A
      CALL  "DPRD_DAT" (
           LADDR                    := W#16#14A,
           RET_VAL                  := "Profibus SFC Alarm".DB3_DBW12,
           RECORD                   := P#DB1.DBX 200.0 BYTE 12);
      CALL  "DPWR_DAT" (
           LADDR                    := W#16#14A,
           RECORD                   := P#DB2.DBX 200.0 BYTE 12,
           RET_VAL                  := "Profibus SFC Alarm".DB3_DBW14);
NETWORK
TITLE = READ/WRITE FROM/TO DRIVE CAGE 18 (ADDRESS 9)
//Dec 342 = Hex 156
      CALL  "DPRD_DAT" (
           LADDR                    := W#16#156,
           RET_VAL                  := "Profibus SFC Alarm".DB3_DBW52,
           RECORD                   := P#DB1.DBX 240.0 BYTE 12);
      CALL  "DPWR_DAT" (
           LADDR                    := W#16#156,
           RECORD                   := P#DB2.DBX 240.0 BYTE 12,
           RET_VAL                  := "Profibus SFC Alarm".DB3_DBW54);
NETWORK
TITLE = READ/WRITE FROM/TO DRIVE CAGE 12 FREFORMING (ADDRESS 10)
//Dec 354 = Hex 162
      CALL  "DPRD_DAT" (
           LADDR                    := W#16#162,
           RET_VAL                  := "Profibus SFC Alarm".DB3_DBW20,
           RECORD                   := P#DB1.DBX 280.0 BYTE 12);
      CALL  "DPWR_DAT" (
           LADDR                    := W#16#162,
           RECORD                   := P#DB2.DBX 280.0 BYTE 12,
           RET_VAL                  := "Profibus SFC Alarm".DB3_DBW22);
NETWORK
TITLE = READ/WRITE FROM/TO DRIVE CAGE 12 (ADDRESS 11)
//Dec 366 = Hex 16E
      CALL  "DPRD_DAT" (
           LADDR                    := W#16#16E,
           RET_VAL                  := "Profibus SFC Alarm".DB3_DBW56,
           RECORD                   := P#DB1.DBX 320.0 BYTE 12);
      CALL  "DPWR_DAT" (
           LADDR                    := W#16#16E,
           RECORD                   := P#DB2.DBX 320.0 BYTE 12,
           RET_VAL                  := "Profibus SFC Alarm".DB3_DBW58);
NETWORK
TITLE = READ/WRITE FROM/TO DRIVE CAGE 6 (ADDRESS 12)
//Dec 378 = Hex 17A
      CALL  "DPRD_DAT" (
           LADDR                    := W#16#17A,
           RET_VAL                  := "Profibus SFC Alarm".DB3_DBW60,
           RECORD                   := P#DB1.DBX 360.0 BYTE 12);
      CALL  "DPWR_DAT" (
           LADDR                    := W#16#17A,
           RECORD                   := P#DB2.DBX 360.0 BYTE 12,
           RET_VAL                  := "Profibus SFC Alarm".DB3_DBW62);
END_FUNCTION

FUNCTION "Take-up traverse alarms" : VOID	// FC 4
TITLE = TAKE-UP TRAVERSE ALARMS FUNCTION
AUTHOR : Milesi
VERSION : 0.1
BEGIN
NETWORK
TITLE = TAKE-UP TRAVERSE MOTOR DRIVE PROFIBUS SLAVE 3 FAULT
      A(;
      L     "MB304";
      L     3;
      ==I;
      );
      AN    "M300.5";
      S     "Db Plc <=> HMI".PROFIBUS.DB100_DBX101_0;
NETWORK
TITLE = TAKE-UP TRAVERSE DRIVEN PINTLE EMERGENCY
      A     "T0";
      AN    "MAP_DI".DB91_DBX007_5;
      AN    "Db Plc <=> HMI".TAKE_UP_1.DB100_DBX107_0;
      S     "Db Plc <=> HMI".TRAVERSE.DB100_DBX105_0;
NETWORK
TITLE = TAKE-UP TRAVERSE IDLE PINTLE EMERGENCY
      A     "T0";
      AN    "MAP_DI".DB91_DBX007_4;
      AN    "Db Plc <=> HMI".TAKE_UP_1.DB100_DBX107_0;
      S     "Db Plc <=> HMI".TRAVERSE.DB100_DBX105_1;
NETWORK
TITLE = TAKE-UP TRAVERSE MOTOR BLOWER OVERLOAD
      A     "T0";
      A     "MAP_DI".DB91_DBX008_6;
      AN    "Db Plc <=> HMI".TAKE_UP_1.DB100_DBX107_0;
      S     "Db Plc <=> HMI".TRAVERSE.DB100_DBX105_2;
NETWORK
TITLE = TAKE-UP TRAVERSE MOTOR DRIVE FAULT
      A     "T0";
      A     "Drives --> Plc".TRVERSE_STATUS_W1.DB1_DBX1_3;
      S     "Db Plc <=> HMI".TRAVERSE.DB100_DBX105_3;
NETWORK
TITLE = TAKE-UP TRAVERSE GENERAL ALARMS
      AN    "Db Plc <=> HMI".PROFIBUS.DB100_DBX101_0;
      AN    "Db Plc <=> HMI".TRAVERSE.DB100_DBX105_0;
      AN    "Db Plc <=> HMI".TRAVERSE.DB100_DBX105_1;
      AN    "Db Plc <=> HMI".TRAVERSE.DB100_DBX105_2;
      AN    "Db Plc <=> HMI".TRAVERSE.DB100_DBX105_3;
      =     "M195.0";
END_FUNCTION

FUNCTION "Take-up traverse unit" : VOID	// FC 5
TITLE = TAKE-UP TRAVERSE UNIT FUNCTION
AUTHOR : Milesi
VERSION : 0.1
BEGIN
NETWORK
TITLE = TAKE-UP TRAVERSE LEFT QUICK JOG
      A(;
      O     "MAP_DI".DB91_DBX008_0;
      O     "MAP_DI".DB91_DBX008_2;
      );
      A     "MAP_DI".DB91_DBX007_5;
      AN    "M182.2";
      AN    "Db Plc <=> HMI".TRAVERSE.DB100_DBX105_3;
      =     "M182.1";
NETWORK
TITLE = TAKE-UP TRAVERSE RIGHT QUICK JOG
      A(;
      O     "MAP_DI".DB91_DBX008_1;
      O     "MAP_DI".DB91_DBX008_3;
      );
      A     "MAP_DI".DB91_DBX007_4;
      AN    "M182.1";
      AN    "Db Plc <=> HMI".TRAVERSE.DB100_DBX105_3;
      =     "M182.2";
NETWORK
TITLE = TAKE-UP TRAVERSE NEGATIVE HOME POSITIONING
      A     "Take-up traverse".HMI_Bit.DB5_DBX1_2;
      AN    "M183.0";
      A     "MAP_DI".DB91_DBX007_4;
      A     "MAP_DI".DB91_DBX007_5;
      A(;
      L     "Take-up traverse".DB5_DBD32;
      L     "Take-up traverse".DB5_DBD24;
      >R;
      );
      S     "M182.4";
      A(;
      O(;
      L     "Take-up traverse".DB5_DBD32;
      L     "Take-up traverse".DB5_DBD24;
      <R;
      );
      ON    "MAP_DI".DB91_DBX007_4;
      ON    "MAP_DI".DB91_DBX007_5;
      ON    "MAP_DI".DB91_DBX004_2;
      ON    "MAP_DI".DB91_DBX000_1;
      ON    "M20.7";
      ON    "M21.0";
      );
      A     "M182.4";
      R     "M182.4";
      NOP   0;
NETWORK
TITLE = TAKE-UP TRAVERSE POSITIVE HOME POSITIONING
      A     "Take-up traverse".HMI_Bit.DB5_DBX1_2;
      AN    "M183.0";
      A     "MAP_DI".DB91_DBX007_4;
      A     "MAP_DI".DB91_DBX007_5;
      A(;
      L     "Take-up traverse".DB5_DBD32;
      L     "Take-up traverse".DB5_DBD24;
      <R;
      );
      S     "M182.3";
      A(;
      O(;
      L     "Take-up traverse".DB5_DBD32;
      L     "Take-up traverse".DB5_DBD24;
      >R;
      );
      ON    "MAP_DI".DB91_DBX007_4;
      ON    "MAP_DI".DB91_DBX007_5;
      ON    "MAP_DI".DB91_DBX004_2;
      ON    "MAP_DI".DB91_DBX000_1;
      ON    "M20.7";
      ON    "M21.0";
      );
      A     "M182.3";
      R     "M182.3";
      NOP   0;
NETWORK
TITLE = TAKE-UP TRAVERSE HOME POSITIONING RUN
      O     "M182.3";
      O     "M182.4";
      =     "M182.5";
      =     "Take-up traverse".HMI_Bit.DB5_DBX0_2;
NETWORK
TITLE = TAKE-UP TRAVERSE RUN
      A(;
      A     "M183.0";
      A     "M180.1";
      A     "Drives --> Plc".BOBBIN_STATUS_W1.DB1_DBX40_2;
      AN    "M10.2";
      O     "M182.5";
      );
      A     "M195.0";
      =     "M182.0";
NETWORK
TITLE = TAKE-UP TRAVERSE DRIVE RUN
      O     "M182.1";
      O     "M182.2";
      O     "M182.0";
      O     "T10";
      =     "Plc --> Drives".TRAVERSE_CONTROL_W1.DB2_DBX1_0;
      =     "Plc --> Drives".TRAVERSE_CONTROL_W1.DB2_DBX1_3;
NETWORK
TITLE = TAKE-UP TRAVERSE ENABLE DELAY TIMER
      A(;
      O     "M182.1";
      O     "M182.2";
      O     "M182.0";
      );
      L     S5T#500MS;
      SF    "T10";
      NOP   0;
      NOP   0;
      NOP   0;
      NOP   0;
NETWORK
TITLE = TAKE-UP TRAVERSE MOTOR BLOWER
      A     "Plc --> Drives".TRAVERSE_CONTROL_W1.DB2_DBX1_0;
      AN    "Db Plc <=> HMI".TRAVERSE.DB100_DBX105_2;
      =     "MAP_DO".DB93_DBX005_0;
NETWORK
TITLE = TAKE-UP TRAVERSE SPEED REFERENCE
//Max Lay = 85 mm
//Max Bobbin rpm = 30.31
//
//(Max Lay * Max Bobbin rpm) * K = 16384
//
//              16384                16384
//K = -------------------------- = ---------- = 6.35938
//    (Max Lay * Max Bobbin rpm)   85 * 30.31
      L     "Take-up traverse".DB5_DBD20;
      L     "Take-up".DB7_DBD40;
      *R;
      L     6.359380e+00;
      *R;
      T     "Take-up traverse".DB5_DBD36;
NETWORK
TITLE = TAKE-UP TRAVERSE SPEED REFERENCE INVERSION
// (network holds code this reader does not know; not shown)
NETWORK
TITLE = TAKE-UP TRAVERSE LEFT QUICK JOG SPEED REFERENCE
      A     "M182.1";
      JNB   J002;
      L     -1.638400e+04;
      T     "Take-up traverse".DB5_DBD36;
J002: NOP   0;
NETWORK
TITLE = TAKE-UP TRAVERSE RIGHT QUICK JOG SPEED REFERENCE
      A     "M182.2";
      JNB   J003;
      L     1.638400e+04;
      T     "Take-up traverse".DB5_DBD36;
J003: NOP   0;
NETWORK
TITLE = TAKE-UP TRAVERSE LEFT HOME POSITIONING SPEED REFERENCE
      A     "M182.4";
      JNB   J004;
      L     -4.096000e+03;
      T     "Take-up traverse".DB5_DBD36;
J004: NOP   0;
NETWORK
TITLE = TAKE-UP TRAVERSE RIGHT HOME POSITIONING SPEED REFERENCE
      A     "M182.3";
      JNB   J005;
      L     4.096000e+03;
      T     "Take-up traverse".DB5_DBD36;
J005: NOP   0;
NETWORK
TITLE = TAKE-UP TRAVERSE SPEED REFERENCE ENABLE
      A     "M182.0";
      A     "MAP_DI".DB91_DBX007_4;
      A     "MAP_DI".DB91_DBX007_5;
      AN    "M10.2";
      O     "M182.1";
      O     "M182.2";
      JC    J006;
      L     0.000000e+00;
      T     "Take-up traverse".DB5_DBD36;
J006: NOP   0;
NETWORK
TITLE = TAKE-UP TRAVERSE MOTOR SPEED REFERENCE TO DRIVE
      L     "Take-up traverse".DB5_DBD36;
      RND;
      T     "Plc --> Drives".DB2_DBW4;
NETWORK
TITLE = TAKE-UP TRAVERSE INVERSION DELAY
      A(;
      A(;
      O(;
      L     "Take-up traverse".DB5_DBD32;
      L     "Take-up traverse".DB5_DBD28;
      <=R;
      );
      O(;
      L     "Take-up traverse".DB5_DBD32;
      L     "Take-up traverse".DB5_DBD24;
      >=R;
      );
      );
      FP    "M10.4";
      S     "M10.2";
      A     "M10.2";
      A(;
      L     "Take-up traverse".DB5_DBD52;
      L     "Take-up traverse".DB5_DBD48;
      >=R;
      );
      R     "M10.2";
      A     "M10.2";
      );
      NOT;
      JNB   J007;
      L     0.000000e+00;
      T     "Take-up traverse".DB5_DBD52;
J007: NOP   0;
NETWORK
TITLE =
      A     "M10.2";
      A     "MAP_DI".DB91_DBX008_5;
      FP    "M10.3";
      JNB   J008;
      L     "Take-up traverse".DB5_DBD52;
      L     1.000000e+00;
      +R;
      T     "Take-up traverse".DB5_DBD52;
J008: NOP   0;
NETWORK
TITLE = TAKE-UP TRAVERSE SPEED REFERENCE LEFT INVERSION BIT
      A(;
      L     "Take-up traverse".DB5_DBD32;
      L     "Take-up traverse".DB5_DBD24;
      >=R;
      );
      O     "Take-up traverse".HMI_Bit.DB5_DBX1_0;
      O     "MAP_DI".DB91_DBX008_0;
      O     "MAP_DI".DB91_DBX008_2;
      R     "M10.1";
NETWORK
TITLE = TAKE-UP TRAVERSE SPEED REFERENCE RIGHT INVERSION BIT
      A(;
      L     "Take-up traverse".DB5_DBD32;
      L     "Take-up traverse".DB5_DBD28;
      <=R;
      );
      O     "Take-up traverse".HMI_Bit.DB5_DBX1_1;
      O     "MAP_DI".DB91_DBX008_1;
      O     "MAP_DI".DB91_DBX008_3;
      S     "M10.1";
NETWORK
TITLE = TAKE-UP TRAVERSE LEFT INVERSION PILOT LAMPS TO HMI
      A     "T0";
      AN    "M10.1";
      =     "MAP_DO".DB93_DBX004_6;
      =     "MAP_DO".DB93_DBX006_0;
NETWORK
TITLE = TAKE-UP TRAVERSE RIGHT INVERSION PILOT LAMPS TO HMI
      A     "T0";
      A     "M10.1";
      =     "MAP_DO".DB93_DBX004_7;
      =     "MAP_DO".DB93_DBX006_1;
NETWORK
TITLE = TAKE-UP TRAVERSE MOTOR RPM TO HMI
      L     "Drives --> Plc".DB1_DBW6;
      ITD;
      DTR;
      L     1.638400e+04;
      /R;
      L     1.420000e+03;
      *R;
      T     "Take-up traverse".DB5_DBD188;
NETWORK
TITLE = TAKE-UP TRAVERSE MOTOR CURRENT TO HMI
      L     "Drives --> Plc".DB1_DBW8;
      ITD;
      DTR;
      L     1.638400e+04;
      /R;
      L     2.550000e+00;
      *R;
      T     "Take-up traverse".DB5_DBD192;
NETWORK
TITLE = TAKE-UP TRAVERSE MOTOR VOLTAGE TO HMI
      L     "Drives --> Plc".DB1_DBW10;
      ITD;
      DTR;
      L     1.638400e+04;
      /R;
      L     4.000000e+02;
      *R;
      T     "Take-up traverse".DB5_DBD196;
END_FUNCTION

FUNCTION "Take-up alarms" : VOID	// FC 6
TITLE = TAKE-UP ALARMS FUNCTION
AUTHOR : Milesi
VERSION : 0.1
BEGIN
NETWORK
TITLE = TAKE-UP BOBBIN MOTOR DRIVE PROFIBUS SLAVE 4 FAULT
      A(;
      L     "MB304";
      L     4;
      ==I;
      );
      AN    "M300.5";
      S     "Db Plc <=> HMI".PROFIBUS.DB100_DBX101_1;
NETWORK
TITLE = TAKE-UP UNIT ET200S PROFIBUS SLAVE 20 FAULT
      A(;
      L     "MB304";
      L     20;
      ==I;
      );
      AN    "M300.5";
      S     "Db Plc <=> HMI".PROFIBUS.DB100_DBX100_4;
NETWORK
TITLE = TAKE-UP 24VDC POWER SUPPLY OVERLOAD 
      A     "T0";
      AN    "MAP_DI".DB91_DBX009_3;
      =     "Db Plc <=> HMI".TAKE_UP_1.DB100_DBX107_0;
NETWORK
TITLE = TAKE-UP 230VAC POWER SUPPLY OVERLOAD 
      A     "T0";
      AN    "MAP_DI".DB91_DBX009_2;
      =     "Db Plc <=> HMI".TAKE_UP_1.DB100_DBX107_1;
NETWORK
TITLE = TAKE-UP BOBBIN MOTOR DRIVE FAULT
      A     "T0";
      A     "Drives --> Plc".BOBBIN_STATUS_W1.DB1_DBX41_3;
      S     "Db Plc <=> HMI".TAKE_UP_1.DB100_DBX107_6;
NETWORK
TITLE = TAKE-UP BOBBIN MOTOR OVERTEMPERATURE
      A     "T0";
      A     "Drives --> Plc".BOBBIN_STATUS_W2.DB1_DBX42_1;
      S     "Db Plc <=> HMI".TAKE_UP_1.DB100_DBX107_5;
NETWORK
TITLE = TAKE-UP AC MOTORS OVERLOAD 
      A     "T0";
      A     "MAP_DI".DB91_DBX009_1;
      AN    "Db Plc <=> HMI".TAKE_UP_1.DB100_DBX107_0;
      =     "Db Plc <=> HMI".TAKE_UP_1.DB100_DBX107_2;
NETWORK
TITLE = TAKE-UP BOBBIN MOTOR BLOWER OVERLOAD
      A     "T0";
      A     "MAP_DI".DB91_DBX004_4;
      AN    "Db Plc <=> HMI".TAKE_UP_1.DB100_DBX107_0;
      =     "Db Plc <=> HMI".TAKE_UP_1.DB100_DBX107_3;
NETWORK
TITLE = TAKE-UP BOBBIN MOTOR ELECTRIC BRAKE OVERLOAD
      A     "T0";
      A     "MAP_DI".DB91_DBX004_5;
      =     "Db Plc <=> HMI".TAKE_UP_1.DB100_DBX107_4;
NETWORK
TITLE = TAKE-UP BOBBIN STOP SERIES PUSH-BUTTON
      A     "T0";
      AN    "MAP_DI".DB91_DBX004_2;
      AN    "M180.1";
      AN    "M183.0";
      AN    "Db Plc <=> HMI".TAKE_UP_1.DB100_DBX107_0;
      =     "Db Plc <=> HMI".TAKE_UP_1.DB100_DBX107_7;
NETWORK
TITLE = TAKE-UP BOBBIN DOWN
      A     "T0";
      A     "M180.1";
      A(;
      ON    "MAP_DI".DB91_DBX006_0;
      ON    "MAP_DI".DB91_DBX006_2;
      );
      AN    "Db Plc <=> HMI".TAKE_UP_1.DB100_DBX107_0;
      S     "M170.0";
NETWORK
TITLE =
      A     "T0";
      A(;
      ON    "MAP_DI".DB91_DBX006_0;
      ON    "MAP_DI".DB91_DBX006_2;
      O     "M170.0";
      );
      AN    "Db Plc <=> HMI".TAKE_UP_1.DB100_DBX107_0;
      =     "Db Plc <=> HMI".TAKE_UP_1.DB100_DBX106_0;
NETWORK
TITLE = TAKE-UP BOBBIN OFF
      A     "T0";
      AN    "M183.0";
      AN    "Db Plc <=> HMI".TAKE_UP_1.DB100_DBX107_0;
      =     "Db Plc <=> HMI".TAKE_UP_1.DB100_DBX106_1;
NETWORK
TITLE = TAKE-UP BOBBIN GENERAL ALARM
      AN    "Db Plc <=> HMI".PROFIBUS.DB100_DBX101_1;
      AN    "Db Plc <=> HMI".PROFIBUS.DB100_DBX100_4;
      AN    "Db Plc <=> HMI".TAKE_UP_1.DB100_DBX106_0;
      AN    "Db Plc <=> HMI".TAKE_UP_1.DB100_DBX107_0;
      AN    "Db Plc <=> HMI".TAKE_UP_1.DB100_DBX107_1;
      AN    "Db Plc <=> HMI".TAKE_UP_1.DB100_DBX107_2;
      AN    "Db Plc <=> HMI".TAKE_UP_1.DB100_DBX107_3;
      AN    "Db Plc <=> HMI".TAKE_UP_1.DB100_DBX107_4;
      AN    "Db Plc <=> HMI".TAKE_UP_1.DB100_DBX107_5;
      AN    "Db Plc <=> HMI".TAKE_UP_1.DB100_DBX107_6;
      AN    "Db Plc <=> HMI".TAKE_UP_1.DB100_DBX107_7;
      =     "M195.1";
END_FUNCTION

